				fbWriteEventData_Day(
					bExecute				:= bWriteData,
					sNetId					:= stFileSetupDayFile.sNetId,
					sPathName				:= stFileSetupDayFile.sTotalName,
					dwTransferBufferStartAdr:= dwTransferBufferStartAdr,
					iNewValues				:= (iIdx-1),
					udNumberofValues		:= udNumberofValues,
					udArrDataSize			:= udArrDataSize,
					udNumberOfEventDatas	:= udNumberOfEventDatas,
					sHeaderOfEventData		:= sHeaderOfEventData,
					eDataType				:= eDataType,
					bBusy					=> ,
					bDone					=> ,
					bError					=> bError,
					nErrId					=> nErrId );
				bWriteDayFileCopy		:= TRUE;
			ELSE
				bWriteDayFileCopy		:= FALSE;
			END_IF

			bWriteData := FALSE;
			state := 1;
		END_IF

		1:
		(* wait for the entries to be written *)
		fbWriteEventData( nNextPointerLoc:= nNextPointerLoc,);
		IF bWriteDayFileCopy THEN
			fbWriteEventData_Day( );
		END_IF
		IF NOT fbWriteEventData.bBusy
	           AND ( (bWriteDayFileCopy AND NOT fbWriteEventData_Day.bBusy) OR NOT bWriteDayFileCopy)
		    THEN
			fbWriteEventData( bExecute:= FALSE,nNextPointerLoc	:= nNextPointerLoc,);
			fbWriteEventData_Day(bExecute := FALSE);

			(*==========================================================*)
			(*  Counter for diagnostic   *)
			(*==========================================================*)
			rTrigErrorWriteData1(CLK:=fbWriteEventData.bError);
			IF rTrigErrorWriteData1.Q THEN
				iErrCounterEventData := iErrCounterEventData + 1;
			END_IF
			rTrigErrorWriteData2(CLK:=fbWriteEventData_Day.bError);
			IF rTrigErrorWriteData2.Q THEN
				iErrCounterEventData_Day := iErrCounterEventData_Day + 1;
			END_IF


			IF NOT fbWriteEventData.bBusy
			    AND ( (bWriteDayFileCopy AND NOT fbWriteEventData_Day.bError) OR NOT bWriteDayFileCopy)
	                  THEN
				(* discard the values already written in file from transfer buffer;
				    move the next values up to the first memory place [first place in the second memory part],make space for later entries *)
				udValuesNotWritten := iIdx-1-fbWriteEventData.udValuesWritten;
				MEMMOVE(
					dwTransferBufferStartAdr,
					dwTransferBufferStartAdr+(fbWriteEventData.udValuesWritten * iOneEntrySize) ,
					udValuesNotWritten * iOneEntrySize);
				(* clear the later space after the values are not written *)

				MEMSET(
					dwTransferBufferStartAdr+(udValuesNotWritten * iOneEntrySize),
					00,
					(udNumberofValues - 1 - udValuesNotWritten) * iOneEntrySize);

	iIdx := iIdx - UDINT_TO_INT(fbWriteEventData.udValuesWritten);
				state := 0;
			END_IF

			IF  NOT fbWriteEventData.bBusy AND NOT  fbWriteEventData.bBusy AND
		 	     NOT	fbWriteEventData.bError AND NOT fbWriteEventData_Day.bError THEN
				state := 0;
			ELSIF (fbWriteEventData.bError OR fbWriteEventData_Day.bError) THEN
				bError:=TRUE;
				state := 0;
			END_IF
		END_IF

	END_CASE


	(*==========================================================*)
	(*  Write to Novram  *)
	(*==========================================================*)
(*	IF NOT bInitNovRAM  AND gbEmbeddedHardwareDetected THEN											(*NEEDED?*)
	
		strucToNOVRAM.iRingBuffer_NextPointerLocation:= nNextPointerLoc;

	END_IF
*)
(*=========== END OF FUNCTION_BLOCK / PROGRAMM =============*)

ACTION M_AddEvent:
IF bInit THEN
	M1_Init( );
END_IF

(* Perform various checks *)
M2_Check( );

(* if no error and trigger event then add the entries *)
IF NOT bInitError AND bTrigEvent
THEN
	iNewValues := iNewValues + 1;		(* count the number of new entries added *)
	IF udCurrentAddIndex = 0 THEN
		udCurrentAddIndex := 1;			(* current index; where the newest entry is located *)
	ELSE
		udCurrentAddIndex := udCurrentAddIndex + 1;
		IF udCurrentAddIndex > udNumberofValues THEN (* current index; wrap around if max reached *)
			udCurrentAddIndex := 1;
		END_IF
	END_IF
	IF udCounter < udNumberOfValues THEN
		udUsedVal := udUsedVal + 1;			(* used index; the number of used entries; once udNumberOfValues reached remains constant to udNumberOfValues *)
	ELSE
		udUsedVal := udNumberofValues;
	END_IF

	IF udUsedVal < udNumberofValues THEN
		udOldestAddIndex := 1;				(* oldest index; wrap around if max reached *)
	ELSIF udUsedVal = udNumberofValues THEN
		udOldestAddIndex := udCurrentAddIndex + 1;
		IF udOldestAddIndex > udNumberofValues THEN		(* oldest index; where the oldest entry is located *)
			udOldestAddIndex := udOldestAddIndex - udNumberofValues;
		END_IF
	END_IF

(*========================================================================*)
(*		 limit description to    STRING[guiKeyAndTextLen];						   *)
(*		 max using length is [uiKeyAndTextLen - sKeySize]                                                     *)
(*=========================================================================*)
	sKeyAndText 			:= CONCAT(sTrigEventKey,'   ');  (* 3 spaces *)
	uiLENsTrigEventText 	:= LEN(sTrigEventText);
	uiLENsMaxText 		:= SIZEOF(sTrigEventText) - LEN(sKeyAndText);
	IF (uiLENsTrigEventText>uiLENsMaxText) THEN
		sTrigEventText := MID(sTrigEventText,0,uiLENsMaxText);
	END_IF
	sKeyAndText := CONCAT(sKeyAndText,sTrigEventText);

	iAddOffset := UDINT_TO_INT(udCurrentAddIndex-1) * iOneEntrySize; (* calculate the offset to be added according to the current index number *)

(*========================================================================*)
(*     fuse the key and text for trigger event together into one string, copy other values        *)
(*========================================================================*)
	(* Add the entry into the buffer *)
	(* Timestamp ------------------------------------- *)

	MEMCPY(dwBufferStartAdr + iAddOffset,ADR(sTimeStamp),SIZEOF(sTimeStamp));
	iSizeOf 			:= SIZEOF(sTimeStamp);
	iAddOffset 		:= iAddOffset + iSizeOf;
	uiCheckEntryLength:= iSizeOf; 					(* check entry length *)

	(* Key and the description -------------------- *)
	MEMCPY(dwBufferStartAdr + iAddOffset,ADR(sKeyAndText),SIZEOF(sKeyAndText));
	iSizeOf 			:= SIZEOF(sKeyAndText);
	iAddOffset 		:= iAddOffset + iSizeOf;
	uiCheckEntryLength:= uiCheckEntryLength + iSizeOf; 	(* check entry length *)

	(* User name --------------------------------------- *)
	MEMCPY(dwBufferStartAdr + iAddOffset,ADR(sUserName),SIZEOF(sUserName));
	iSizeOf 			:= SIZEOF(sUserName);
	iAddOffset 		:= iAddOffset + iSizeOf;
	uiCheckEntryLength:= uiCheckEntryLength + iSizeOf; 	(* check entry length *)

	(* Brake program --------------------------------------- *)
	MEMCPY(dwBufferStartAdr + iAddOffset,ADR(sBrakeProgram),SIZEOF(sBrakeProgram));
	iSizeOf 			:= SIZEOF(sBrakeProgram);
	iAddOffset 		:= iAddOffset + iSizeOf;
	uiCheckEntryLength:= uiCheckEntryLength + iSizeOf; 	(* check entry length *)



(*========================================================================*)
(*				 process value for logging only for real-type                                                  *)
(*=========================================================================*)
	(* copy the event datas into memory *)
	FOR i := 1 TO iNumberOfEventDatas DO

		CASE eDataType[i] OF
			(* Delete other type of data*)


			eReal :

				MEMCPY(dwBufferStartAdr + iAddOffset, dwArrDataAdr[i], udArrDataSize[i]);
				ar_iAddOffset[i] := iAddOffset;
				iAddOffset := iAddOffset + UDINT_TO_INT(udArrDataSize[i]);

		END_CASE


		iSizeOf 		:= UDINT_TO_INT(udArrDataSize[i]);
		uiCheckEntryLength:= uiCheckEntryLength + iSizeOf; 	(* check entry length *)

	END_FOR

(*========================================================================*)
(*				 Check length of data and the buffer entry size in the array		              *)
(*=========================================================================*)
	IF (uiCheckEntryLength>iOneEntrySize ) THEN
		uiCheckLenghtError := uiCheckLenghtError + 1;
		strLastKeyError := sKeyAndText;
	END_IF

	bCheck := TRUE;
END_IF
END_ACTION

ACTION M_CheckEvent:
(* At the end of the PLC cycle Check the data and order in ascending sequence *)
IF bCheck THEN (* bcheck is set to true by M_AddEvent; which means when no events or M_AddEvent not called, no data exists and hence no check performed *)

	iNumberOfValues := UDINT_TO_INT(udNumberofValues);		(* copy udint into int form *)

	(* if fill the buffer from beginning then reset the whole buffer *)
	IF iIdx = 1 THEN
		MEMSET(dwTransferBufferStartAdr,00,udSizeOfeachBlock);		(* reset the buffer *)
	END_IF

	(* see if all the new values fit into transfer buffer, else reassign New values to fitting number of values *)
	IF (iIdx + iNewValues) > (iNumberOfValues - 1) THEN
		iNewValues := (iNumberOfValues - 1) - iIdx;
	END_IF

	(* Copy the entries into transfer buffer *)
	IF udCurrentAddIndex >= iNewValues THEN 				(* If current index went once round the ring and is less then the new events added, which means some new events at the end of Ring Buffer and some in the beginning *)
		(* if New values are less than the current index that means all the values are in the beginning *)
		MEMCPY(
			dwTransferBufferStartAdr+((iIdx-1)*iOneEntrySize),
			dwBufferStartAdr+((udCurrentAddIndex - iNewValues)*iOneEntrySize),
			iNewValues*iOneEntrySize);


	ELSE
		(* if new values is greater than the current index that means some are at the end and rest in the beginning of the bufffer *)
		udOldValuesToBeCopied := iNewValues - udCurrentAddIndex;

		MEMCPY(
			dwTransferBufferStartAdr+((iIdx-1)*iOneEntrySize),
			dwBufferStartAdr+((udNumberofValues - udOldValuesToBeCopied)*iOneEntrySize),
			udOldValuesToBeCopied*iOneEntrySize);

		MEMCPY(
			dwTransferBufferStartAdr+((iIdx-1+udOldValuesToBeCopied)*iOneEntrySize),
			dwBufferStartAdr,
			udCurrentAddIndex*iOneEntrySize);
	END_IF

(*========================================================================*)
(*                                                      to sort out key number                                                                      *)
(*========================================================================*)
(*																									(*WIESO ausgeklammert?*)
	jIdx := iIdx;
	FOR i := iIdx TO (iIdx - 1 + iNewValues) DO		(* for loop from new index value to the number of new values *)

		MEMCPY(
			ADR(sKeyAndText_1),
			dwTransferBufferStartAdr+((i-1)*iOneEntrySize)+ SIZEOF(sTimeStamp),
			SIZEOF(sTrigEvent));

		sKeyAndText_1 := LEFT (sKeyAndText_1,(FIND(sKeyAndText_1,'   '))-1); (*01_05_001*)
		sKeyAndText_1 := DELETE (sKeyAndText_1,1,3);(*0105_001*)
		sKeyAndText_1 := DELETE (sKeyAndText_1,1,5); (*0105001*)
		udKeyAndText_1 := STRING_TO_UDINT(sKeyAndText_1);
		(* Arrange the key in an ascending order *)
		FOR j := jIdx TO (jIdx -1 + iNewValues) DO
			MEMCPY(
				ADR(sKeyAndText_2),
				dwTransferBufferStartAdr+((j-1)*iOneEntrySize)+SIZEOF(sTimeStamp),
				SIZEOF(sTrigEvent));

			sKeyAndText_2 := LEFT (sKeyAndText_2,(FIND(sKeyAndText_2,'   '))-1); (*01_05_001*)
			sKeyAndText_2 := DELETE (sKeyAndText_2,1,3);(*0105_001*) (* delete underscore *)
			sKeyAndText_2 := DELETE (sKeyAndText_2,1,5); (*0105001*) (* delete underscore *)
			udKeyAndText_2 := STRING_TO_INT(sKeyAndText_2);	(* convert string to a number for the necessary checks to sort *)
			IF udKeyAndText_1 < udKeyAndText_2 THEN
				(* use last memory address as temp memory space for comparison *)
				MEMCPY(
					dwTransferBufferStartAdr+((iNumberOfValues-1)*iOneEntrySize),
					dwTransferBufferStartAdr+((j-1)*iOneEntrySize),
					iOneEntrySize);
				MEMCPY(
					dwTransferBufferStartAdr+((j-1)*iOneEntrySize),
					dwTransferBufferStartAdr+((i-1)*iOneEntrySize),
					iOneEntrySize);
				MEMCPY(
					dwTransferBufferStartAdr+((i-1)*iOneEntrySize),
					dwTransferBufferStartAdr +((iNumberOfValues-1)*iOneEntrySize),
					iOneEntrySize);

				udKeyAndText_1 := udKeyAndText_2;			(*exchange the strings *)
			END_IF
		END_FOR
	END_FOR
	(*========================================================================*)
	(*                                                 end  to sort out key number                                                                  *)
	(*========================================================================*)
*)
	bCheck := FALSE;			(* Checking done *)
	iIdx := iIdx + iNewValues;	(* calculate where the index stands; increment the value of index by number of new values *)

	iEntriesWritten := iEntriesWritten + iNewValues;		(* Count the number of entries written *)
	IF iEntriesWritten > udNumberofValues THEN				(* If overflow then calculate relative count *)
		iEntriesWritten := UDINT_TO_INT(udNumberofValues - INT_TO_UDINT(iEntriesWritten));
	END_IF

	IF (iIdx-1) > 0 AND state = 0 THEN
		bWriteData := TRUE;
	END_IF
	iNewValues := 0;				(* reset the new values counter to zero *)

END_IF
END_ACTION

ACTION M1_Init:
bInit := FALSE;

iOneEntrySize := 0;				(* size of event in memory *)
iOneEntrySize := 	SIZEOF(sTimeStamp)+
				SIZEOF(sTrigEventText)+  (*before sTrigEvent*)
					SIZEOF(sUserName) +
					SIZEOF(sBrakeProgram);

iOneEntryLength := 0;			(* length of the event when written in file *)
iOneEntryLength :=	SIZEOF(sTimeStamp) +
					LEN(sTab) +
				SIZEOF(sTrigEventText)+  (*before SIZEOF(sTrigEventKey) + SIZEOF(sTrigEventText)+*)
					LEN(sTab) +
					SIZEOF(sUserName) +
					LEN(sTab) +
					SIZEOF(sBrakeProgram) +
					LEN(sTab);

iNumberOfEventDatas := UDINT_TO_INT(udNumberOfEventDatas);

(* Check the data type of all the required event datas; calculate entry length and size accordingly *)
FOR i := 1 TO iNumberOfEventDatas DO
	CASE eDataType[i] OF
		eBool :
			iOneEntryLength := iOneEntryLength + 5;			(* when converted into string *)
			iOneEntrySize := iOneEntrySize +  UDINT_TO_INT(udArrDataSize[i]);

		eReal :
			iOneEntryLength := iOneEntryLength + 17;		(* when converted into string *)
			iOneEntrySize := iOneEntrySize +  UDINT_TO_INT(udArrDataSize[i]);

	END_CASE
	IF i < udNumberOfEventDatas THEN
		iOneEntryLength := iOneEntryLength + LEN(sTab);	(* calculate the tabs too into the length of string *)
	ELSE
		iOneEntryLength := iOneEntryLength + LEN(sLineFeed);	(* calculate the linefeed too into the length of string *)
	END_IF

END_FOR

IF ((udLoggedEventSize/2) MOD iOneEntrySize) = 0 THEN		(* Check if all the data fits into the given memory block *)
	udSizeOfeachBlock := udLoggedEventSize/2;
	udNumberofValues := udLoggedEventSize/ (iOneEntrySize *2);	(* calculate the number of events that can be logged *)
	(* calulate the start and end addresses of the buffer *)
	dwBufferStartAdr := dwLoggedEventAdr;
	dwBufferEndAdr	:= dwLoggedEventAdr + udLoggedEventSize/2;
	dwTransferBufferStartAdr := dwBufferEndAdr;
	dwTransferBufferEndAdr := dwLoggedEventAdr + udLoggedEventSize;
ELSE
	bInitError := TRUE;	(* size not appropriate *)
	nErrId := 1;
END_IF
END_ACTION

ACTION M2_Check:
(* check if the file path is given *)
IF LEN(stFileSetup.sPathName)= 0
THEN
	ADSLOGSTR( 	msgCtrlMask := ADSLOG_MSGTYPE_WARN,
				msgFmtStr := 'PLC Msg: FilePath is empty; %s',
				strArg := stFileSetup.sPathName);
	RETURN;
END_IF
(* check if the file path is given for Day file *)
IF bWriteDayFile AND LEN(stFileSetupDayFile.sPathName)= 0
THEN
	ADSLOGSTR( 	msgCtrlMask := ADSLOG_MSGTYPE_WARN,
				msgFmtStr := 'PLC Msg: FilePath_DayFile is empty; %s',
				strArg := stFileSetupDayFile.sPathName);
	RETURN;
END_IF
(* If same file name for RingBufferFile and for EventDayFile *)
IF bWriteDayFile AND (stFileSetup.sPathName = stFileSetupDayFile.sPathName)
THEN
	ADSLOGSTR( 	msgCtrlMask := ADSLOG_MSGTYPE_WARN,
				msgFmtStr := 'PLC Msg: Same file path given; %s',
				strArg := stFileSetupDayFile.sPathName);
	RETURN;
END_IF

(* Check the start, end addresses of buffers *)
IF dwBufferStartAdr = 0 OR dwBufferEndAdr = 0 OR
   dwTransferBufferStartAdr = 0 OR dwTransferBufferEndAdr = 0
THEN
	ADSLOGDINT( msgCtrlMask := ADSLOG_MSGTYPE_WARN,
				msgFmtStr := 'PLC Msg: Buffer Size does not match; Buffer Addresses zero; %s',
				dintArg := MIN(dwBufferStartAdr,MIN(dwBufferEndAdr,MIN(dwTransferBufferStartAdr,dwTransferBufferEndAdr))));
	RETURN;
END_IF

(* If entry length in file larger than 255, string operations like CONCAT, LEN do not work *)
IF iOneEntryLength > 255
THEN
	ADSLOGDINT( msgCtrlMask := ADSLOG_MSGTYPE_WARN,
				msgFmtStr := 'PLC Msg: Entry of one event is greater 255; %s',
				dintArg := iOneEntryLength);
	RETURN;
END_IF

(* Check the entry size in memory *)
IF iOneEntrySize = 0
THEN
	ADSLOGDINT( msgCtrlMask := ADSLOG_MSGTYPE_WARN,
				msgFmtStr := 'PLC Msg: Buffer size is Zero; %d',
				dintArg := iOneEntrySize);
	RETURN;
END_IF

(* Check if the trigger event key is not empty *)
IF sTrigEventKey = ''
THEN
	ADSLOGSTR( 	msgCtrlMask := ADSLOG_MSGTYPE_WARN,
				msgFmtStr := 'PLC Msg: TrigEventKey is empty; %s',
				strArg := sTrigEventKey);
	RETURN;
END_IF

(* Check if the trigger event key is according to the format*)
IF LEN(sTrigEventKey) < SIZEOF(sTrigEventKey)-1
THEN
	ADSLOGSTR( 	msgCtrlMask := ADSLOG_MSGTYPE_WARN,
				msgFmtStr := 'PLC Msg: TrigEventKey length not as per defined; %s',
				strArg := sTrigEventKey);
	RETURN;
END_IF

(* Check if the Buffer start address is not zero; nonassigned *)
IF dwBufferStartAdr = 0
THEN
	ADSLOGSTR( 	msgCtrlMask := ADSLOG_MSGTYPE_WARN,
				msgFmtStr := 'PLC Msg: Buffer start address is 0; %s',
				strArg := sTrigEventKey);
	RETURN;
END_IF

(* Check if the Buffer end address is not zero; nonassigned *)
IF dwBufferEndAdr = 0
THEN
	ADSLOGSTR( 	msgCtrlMask := ADSLOG_MSGTYPE_WARN,
				msgFmtStr := 'PLC Msg: Buffer end address is 0; %s',
				strArg := sTrigEventKey);
	RETURN;
END_IF

(* Check if the transfer Buffer start address is not zero; nonassigned *)
IF dwTransferBufferStartAdr = 0
THEN
	ADSLOGSTR( 	msgCtrlMask := ADSLOG_MSGTYPE_WARN,
				msgFmtStr := 'PLC Msg: Buffer start address is 0; %s',
				strArg := sTrigEventKey);
	RETURN;
END_IF

(* Check if the transfer Buffer end address is not zero; nonassigned *)
IF dwTransferBufferEndAdr = 0
THEN
	ADSLOGSTR( 	msgCtrlMask := ADSLOG_MSGTYPE_WARN,
				msgFmtStr := 'PLC Msg: Buffer end address is 0; %s',
				strArg := sTrigEventKey);
	RETURN;
END_IF

(* Check if the size of block is nonzero; nonassigned *)
IF udSizeOfeachBlock = 0
THEN
	ADSLOGSTR( 	msgCtrlMask := ADSLOG_MSGTYPE_WARN,
				msgFmtStr := 'PLC Msg: Buffer size is 0; %s',
				strArg := sTrigEventKey);
	RETURN;
END_IF
END_ACTION

END_FUNCTION_BLOCK

// ---- Alarm System/POUs/02_Alarm_Handling/FB_WriteEventData.TcPOU
FUNCTION_BLOCK FB_WriteEventData
(**********************************************************************************)
(**********************************************************************************)
(*  	VERSION:			002.012
							                									
	PROGRAMMED BY:	Puja					  					
  	Changed by:			Hardy Patommel							
*)  																		
(*-----------------------------------------------------------------------------------------------------------------------------------*)
(*  REVISIONS:						                							 
   	Date		|	Version/Author 	|	Remark
	----------------------------------------------------------------------------------------------------
	2007-10-08	|	001.001     HP		|   	formatting the REAL value FOR the file output
	2008-03-04	|	002.000     HP		|   	add header function block
	2008-03-27	|	002.001     HP		|   	add header length with initialization value
	2009-03-26	|	002.010     HP		|   	get header length as parameter
	2009-03-27	|	002.011     HP		|   	change strBuffer size with a constant variable
	2009-08-09	|	002.012     HP		|   	change sTimestamp[24]
*)
(*-----------------------------------------------------------------------------------------------------------------------------------*)
(*  	DESCRIPTION:
	Constant value for the file layout >>	
		nNextPointerLoc			: DINT;		>>> actual position for the next entry [NOVRAM]
		iFirstHeaderLEN1			: INT:=1000;	>>> header size without column-description

	Note:
		 iFirstHeaderLEN and iColumnLineLEN are only necessary when the data file will be create
*)
(**********************************************************************************)
(**********************************************************************************)
VAR_INPUT
	bExecute 				: BOOL;
	sNetId					: T_AmsNetId;
	sPathName				: T_MaxString;
	dwTransferBufferStartAdr	: DWORD;
	iNewValues				: INT;
	udNumberofValues 		: UDINT;
	udNumberOfEventDatas	: UDINT;
	udArrDataSize			: ARRAY [1..NUMBER_OF_EVENT_DATAS] OF UDINT;
	eDataType				: ARRAY [1..NUMBER_OF_EVENT_DATAS] OF E_DataType;
	sHeaderOfEventData	: ARRAY [1..giGeneralLoggerChannelInUsed] OF STRING(giGeneralLenghtOfName);
	iHeaderLEN				: INT;  (*length of whole header; first header + column*)
END_VAR
VAR_IN_OUT
	nNextPointerLoc			: DINT;
END_VAR
VAR_OUTPUT
	udValuesWritten			: UDINT;
	bBusy					: BOOL;
	bDone					: BOOL;
	bError					: BOOL;
	nErrId					: UDINT;
END_VAR
VAR
	RExec_Trig				: R_TRIG;
	hFile					: UINT;
	fbFileOpen				: FB_FileOpen;
	fbFileSeek				: FB_FileSeek;
	fbFileWrite				: FB_FileWrite;
	fbFileClose				: FB_FileClose;
	tAdsTimeOut			: TIME:= T#10s;
	eFileState				: E_FileState_SC;
	nMode					: DWORD;
	sStrBuffer				: STRING(guiStrBufferSize);	(* header 1100 + row 200 * 218 sign = 44700*)
	sStrHeader				: STRING(2170);	 	(*10 row with 217 sign*)
	sVar					: STRING(255);
	sHeader					: STRING(giHeaderColumnLineLEN); (*:='TimeStampUTC$TTrigKey$TUserName$TBrakeProgram$T'; (*!!HP*)		DISABLED BY NIHAL MALIK *)
	sTab					: STRING[2] := '$T';
	sLineFeed				: STRING[4] := '$R$N';

	i						: INT;


	dwCaptureTransferBufferStartAdr : DWORD;
	sTimeStamp			: STRING[24];	(* Time the Statuscode becomes true *)
	sTrigEvent				: STRING[guiKeyAndTextLen];	(* key and Text of Statuscode, like sKeyAndText[80] in M_AddEvent*)
	sUserName				: STRING[24];	(* name of the user who had the Active Status to do the operation *)
	sBrakeProgram			: STRING[4]; 	(* Activated brake program *)
	rVar						: REAL;
(*	eTime					:= 12,
	eDate					:= 13,
	eTime_OF_Day			:= 14,
	eDateAndTime			:= 15,
	eString					:= 16,	*)
	iCopyOffset				: INT;

	iPrepIndex				: INT;
	iStrBufferIdx				: UINT; (*Index buffer*)

	iStrLineIdx				: INT; (*Index line*)
	iStuff					: INT;
	iStartStuffIndex			: INT;
	iEndStuffIndex			: INT;
	iStartIndex				: INT;
	iEndIndex				: INT;

	iBatchValue				: INT := 20;(* in batch of how many entries is the data to be written *)
	iEventsWrittenCurrent		: INT;		(* Event written in current cycle *)
	iCaptureNewValues		: INT;		(* captures new values *)
	iEntriesWritten			: INT;		(* Entries Written; so as to calculate the next pointer location*)
	iFittingEntries				: INT;		(* number of entries fitting *)
	iEventsInCycle			: INT;		(* In how many batches is data written *)
	bHeader					: BOOL;		(* If a new file write then to write the header *)
	iCounter					: INT;		(* Total number of entries written till now, so as to tally *)
	iNumberOfEventDatas		: INT;
	sTimestampShort			: STRING[12];
	sRealDataReduce		: STRING[10];
	iLength					: INT;
	iDiffenzLength				: INT;
	iForIndex					: UINT;

	fbHeaderForLogging		: FB_HeaderForLogging;
	iFirstHeaderLEN			: INT;
	iColumnLineLEN		: INT;
	uiCountsOfLine			: UINT;
	udiCheckHeaderLength	: UDINT;

END_VAR

(*========== START OF FUNCTION_BLOCK / PROGRAMM ============*)


(*=====================================================================*)
(*					write event data to file        							     *)
(*=====================================================================*)
RExec_Trig( CLK := bExecute );

CASE eFileState OF
   eInit_SC:
		IF RExec_Trig.Q THEN	(* Rising edge triggered *)
			bBusy 	:= TRUE;
			bError	:= FALSE;
			bDone 	:= FALSE;
			nErrId	:= 0;
			hFile	:= 0;

			dwCaptureTransferBufferStartAdr := dwTransferBufferStartAdr;(* capture the transfer buffer address *)
			iCaptureNewValues	:= iNewValues;					(* make a copy of the input newvalues *)
			iNumberOfEventDatas := UDINT_TO_INT(udNumberOfEventDatas);
			nMode := FOPEN_MODEREAD OR FOPEN_MODEPLUS OR FOPEN_MODEBINARY;
			(*nMode := FOPEN_MODEAPPEND OR FOPEN_MODEPLUS OR FOPEN_MODEBINARY;*)
			iBatchValue := (guiStrBufferSize/iOneEntryLength) - 1;		(* calculate the batch size in which data is to be written *)
			IF iCaptureNewValues > 0 THEN
				sTimestampShort :='4';(* FUN_TimeToString(Lib_strucSystemTime); (*access time *)TO ACTION*)
				(* Open a file *)
				fbFileOpen( bExecute	:= FALSE	);
				fbFileOpen(	bExecute	:= TRUE,
							sNetId		:= sNetID,
							sPathName	:=sPathName,
							nMode		:= nMode,
							ePath		:= Path_Generic,
							tTimeout	:= tAdsTimeOut );

				eFileState := eFileOpen_SC;
				(* reset the variables *)
				iStartIndex := 1;
				iStrBufferIdx := 0;
				sStrBuffer := '';
				sVar := '';
				udValuesWritten := 0;
			END_IF
		END_IF

		g_TriggSendExeAlarmList := FALSE;

	eFileOpen_SC:	(* Wait for the file to be opened *)
		fbFileOpen( );
		IF NOT fbFileOpen.bBusy THEN
			fbFileOpen(	bExecute := FALSE);

			IF NOT fbFileOpen.bError THEN		(* if no error; File already exists *)

				IF NOT bHeader AND nNextPointerLoc > 0 THEN		(*Check the next pointer persistent value*)
					nNextPointerLoc := nNextPointerLoc -  iHeaderLEN;
					IF  iOneEntryLength <> 0 THEN
						iEntriesWritten := DINT_TO_INT(nNextPointerLoc/iOneEntryLength);
						iCounter := DINT_TO_INT(nNextPointerLoc/iOneEntryLength);
					END_IF

					nNextPointerLoc := nNextPointerLoc + iHeaderLEN;

				ELSIF bHeader THEN		(* if file did not exist then iEntriesWritten to beginning *)
					iEntriesWritten := 0;
					iCounter := 0;
				ELSIF NOT bHeader AND (nNextPointerLoc = 0) THEN	(* reset all and file exist *)
					nNextPointerLoc := nNextPointerLoc + iHeaderLEN;
				END_IF
				iFittingEntries := UDINT_TO_INT(udNumberofValues)  - iEntriesWritten ;
				(* calculate the minimum of Captured values, Batch value and how many can fit *)
				iEndIndex := MIN(iCaptureNewValues,iBatchValue);
				iEventsWrittenCurrent := iEndIndex := MIN(iEndIndex, iFittingEntries);

				hFile  := fbFileOpen.hFile;
				fbFileSeek( bExecute := FALSE);			(* File Seek *)
				fbFileSeek(	sNetId 		:= sNetId,
							hFile		:= hFile,
							nSeekPos	:= nNextPointerLoc,			(* File pointer to zero *)
							eOrigin		:= SEEK_SET,
							bExecute	:= TRUE,
							tTimeout	:= tAdsTimeOut,
							);
				eFileState := eFileSeek_SC;

			ELSE	(*if error, File does not exist; a new file is to be written *)

				(*create new file with header*)
				nMode := FOPEN_MODEWRITE  OR FOPEN_MODEPLUS OR FOPEN_MODEBINARY;
				(*nMode := FOPEN_MODEAPPEND  OR FOPEN_MODEPLUS OR FOPEN_MODEBINARY;*)
				fbFileOpen( bExecute	:= FALSE	);
				fbFileOpen(	bExecute	:= TRUE,
				 			sNetId		:= sNetID,
							sPathName	:= sPathName,
							nMode		:= nMode,
							ePath		:= Path_Generic,
							tTimeout	:= tAdsTimeOut );
				eFileState := eFileOpen_SC;
				nNextPointerLoc := 0;
				iCounter := 0;
				(* if new file is being written then write down the header *)
				bHeader := TRUE;

				fbHeaderForLogging(
						st_TurbineIdent		:= st_xTurbineIdent ,			(*general machine info*)
						s_FileDescription	:= fbSCLogger.stFileSetup.sFileDescription,
						s_ColumnText 		:= gstrRingBufferFileColumnText,
						ar_ColumnText		:= sHeaderOfEventData,		(*array of column description*)
						iCountsOfColumns	:= iNumberOfEventDatas,	(*counts of columns*)
						iOneEntryLength	:= giRingBufferFileOneEntryLength,(*length of every entry, all lines with the same length, see init-logger*)
				//ACTION		adr_sHeader1		:= ADR(sStrHeader) ,		(*part one of the header*)
				//ACTION		adr_sColumnLine	:= ADR(sHeader),			(*part two of the header*)
						iCountsOfLine		=> uiCountsOfLine,			(*lines of the part one header*)
						iHeaderLEN			=> iFirstHeaderLEN,			(*length of the part one header*)
						iColumnLineLEN	=> iColumnLineLEN);		(*length of the part two header*)


				(*Check the header length: header and column-description*)
				udiCheckHeaderLength := LEN(sStrHeader) + LEN(sHeader);
			END_IF
		END_IF


	eFileSeek_SC:
		fbFileSeek( );
		IF NOT fbFileSeek.bBusy THEN
			fbFileSeek(bExecute := FALSE );
			IF NOT fbFileSeek.bError THEN

				(* Prepare the data to be written *)
				M_PrepareWriteData( );

				(* Write into File *)
				fbFileWrite( 	bExecute	:= FALSE	);
				fbFileWrite(  	bExecute	:= TRUE,
								sNetId		:= sNetID,
								hFile		:= hFile,
								pWriteBuff	:= ADR(sStrBuffer),
								cbWriteLen	:= iStrBufferIdx,         (*Write not the whole Buffer, only new entries*)
								tTimeout	:= tAdsTimeOut	);

				iStrBufferIdx := iStrBufferIdx;

				eFileState := eFileWrite_SC;

			ELSE
				bBusy := FALSE;
				bError := TRUE;
				nErrId := fbFileSeek.nErrId;
				eFileState := eInit_SC;
			END_IF
		END_IF


	eFileWrite_SC:	(* Wait until  the file is written *)
		fbFileWrite();
		IF NOT fbFileWrite.bBusy THEN
			fbFileWrite(bExecute := FALSE);
			IF NOT fbFileWrite.bError THEN
				bHeader := FALSE;
				IF iCaptureNewValues > iEventsWrittenCurrent THEN		(* data is to be written into two or more parts *)
					IF iEventsWrittenCurrent = iBatchValue THEN
						(* sStrBuffer was insufficient to occupy all entries, Fitting entries were greater than that, continue writting at same file pointer *)
						iEntriesWritten := iEntriesWritten + iBatchValue;
						iFittingEntries := iFittingEntries - iEventsWrittenCurrent;
						iCaptureNewValues := iCaptureNewValues - iEventsWrittenCurrent;
						iEndIndex := MIN( iCaptureNewValues , iBatchValue);
						iEventsWrittenCurrent := iEndIndex := MIN( iEndIndex , iFittingEntries); (* Events to be written in current write cycle;*)
						iStrBufferIdx := 0;				(* reset while new batch write *)

						(* Prepare the next batch of data to be written *)
						M_PrepareWriteData( );

						(* Write into File *)
						fbFileWrite( 	bExecute	:= FALSE	);
						fbFileWrite(  	bExecute	:= TRUE,
								sNetId		:= sNetID,
								hFile		:= hFile,
								pWriteBuff	:= ADR(sStrBuffer),
								cbWriteLen	:= iStrBufferIdx,         (*Write not the whole Buffer, only new entries*)
								tTimeout	:= tAdsTimeOut	);

						iStrBufferIdx := iStrBufferIdx;
						eFileState := eFileWrite_SC;

					ELSIF iEventsWrittenCurrent = iFittingEntries THEN
						(* if the events written was just fit; pointer location to be set to beginning of file *)
						(* -------------------------------------------------------------------------------------------------------------*)
						iEntriesWritten := 0;
						iFittingEntries := UDINT_TO_INT(udNumberofValues);		(* go to beginning of file and initialise fitting entries to max *)
						iCaptureNewValues := iCaptureNewValues - iEventsWrittenCurrent;
						iEventsWrittenCurrent := iEndIndex := MIN( iCaptureNewValues , iBatchValue);
						iStrBufferIdx := 0;

						(* calculate the next pointer location *)
						nNextPointerLoc := iHeaderLEN + (iEntriesWritten * iOneEntryLength);
						fbFileSeek( bExecute := FALSE);			(* File Seek *)
						fbFileSeek(	sNetId 		:= sNetId,
									hFile		:= hFile,
									nSeekPos	:= nNextPointerLoc,	(* File pointer to next loc - first line in file*)
									eOrigin		:= SEEK_SET,
									bExecute	:= TRUE,
									tTimeout	:= tAdsTimeOut
									);
						eFileState := eFileSeek_SC;
					END_IF

				ELSE	(* if exact fit then reintialise pointer to start of file *)
						(* ------------------------------------------------------------------*)
					IF iFittingEntries = iCaptureNewValues THEN
						iEntriesWritten := 0; (* actually 200 but reset to 1 *)
					ELSE
						iEntriesWritten := iEntriesWritten + iCaptureNewValues;
					END_IF
					nNextPointerLoc :=iHeaderLEN + ( iEntriesWritten * iOneEntryLength);
					(* Close the File *)
					fbFileClose(	bExecute:= FALSE	);
					fbFileClose(	bExecute:= TRUE,
									sNetId	:= sNetID,
									hFile	:= hFile,
									tTimeout:= tAdsTimeOut	);
					eFileState := eFileClose_SC;
				END_IF
			ELSE
				bBusy := FALSE;
				bError := TRUE;
				nErrId := fbFileWrite.nErrId;
				eFileState := eInit_SC;
			END_IF
		END_IF



	eFileClose_SC:	(* Wait untill File is closed *)
		fbFileClose();
		IF NOT fbFileClose.bBusy THEN
			fbFileClose( bExecute:= FALSE );
			IF NOT fbFileClose.bError THEN
				IF iCounter >= UDINT_TO_INT(udNumberOfValues) THEN
					iCounter := iCounter;
				END_IF
				(*eFileState := eInit_SC;*)
				eFileState := eFileCopy_SC;
				bBusy  := FALSE;
				bDone  := TRUE;
				bHeader := FALSE;
				sStrBuffer := '';
				iCaptureNewValues := 0;
				iEventsInCycle := 0;
			ELSE
				bBusy := FALSE;
				bError := TRUE;
				nErrId := fbFileClose.nErrId;
				eFileState := eInit_SC;
			END_IF
		END_IF

		eFileCopy_SC:
			g_TriggSendExeAlarmList := TRUE;
			eFileState := eInit_SC;

END_CASE

(*=========== END OF FUNCTION_BLOCK / PROGRAMM =============*)

ACTION M_PrepareWriteData:
MEMSET(ADR(sStrBuffer) , 0, LEN(sStrBuffer));
IF bHeader  THEN
	(*Header part one*)
	MEMCPY(ADR(sStrBuffer) ,ADR(sStrHeader),iFirstHeaderLEN);
	(*Header part two, column description*)
	MEMCPY(ADR(sStrBuffer)+iFirstHeaderLEN ,ADR(sHeader),iColumnLineLEN);
	(*index for buffer entry after the header; iHeaderLEN := iFirstHeaderLEN + iColumnLineLEN;*)
	iStrBufferIdx := iHeaderLEN;
	(* Write into File *)
END_IF

(* Stuff the data to be written into a string buffer *)
FOR iPrepIndex := iStartIndex  TO iEndIndex DO	(* for loop from new index value to the number of new values *)
	iCopyOffset := (((iPrepIndex-1)+iEventsInCycle)*iOneEntrySize); (*iCopyOffset := Offset in array ringbuffer*)
	sVar := '';
	iStrLineIdx := 0; (*index for the line, function stuff line*)
	(*gets the new dataset ####################*)
	(*gets timestamp value ---------------*)
	MEMCPY(
		ADR(sTimeStamp),
		dwCaptureTransferBufferStartAdr+iCopyOffset,
		SIZEOF(sTimeStamp));
	sVar := CONCAT('',sTimeStamp);
	sVar := CONCAT(sVar,sTab);
	iCopyOffset := iCopyOffset + SIZEOF(sTimeStamp);

	(*gets trigger event string ---------------*)
	MEMCPY(
		ADR(sTrigEvent),
		dwCaptureTransferBufferStartAdr+iCopyOffset,
		SIZEOF(sTrigEvent));
	(*look and fill to 50 sign*)
	iLength := LEN(sTrigEvent);
	IF (iLength<giCountsOfKeyLetterForStatuscodeFile) THEN
		iDiffenzLength := giCountsOfKeyLetterForStatuscodeFile - iLength ;
		FOR iForIndex := 1 TO  iDiffenzLength DO
			sTrigEvent := CONCAT(sTrigEvent,' ');
		END_FOR
	END_IF
	sTrigEvent := sTrigEvent ;
	sVar := CONCAT(sVar,sTrigEvent);
	sVar := CONCAT(sVar,sTab);
	iCopyOffset := iCopyOffset + SIZEOF(sTrigEvent); (*read data out of log-array*)

	(*gets user name string ---------------*)
	MEMCPY(
		ADR(sUserName),
		dwCaptureTransferBufferStartAdr+iCopyOffset,
		SIZEOF(sUserName));
	sVar := CONCAT(sVar,sUserName);
	sVar := CONCAT(sVar,sTab);
	iCopyOffset := iCopyOffset + SIZEOF(sUserName);

	(*gets brake program string ---------------*)
	MEMCPY(
		ADR(sBrakeProgram),
		dwCaptureTransferBufferStartAdr+iCopyOffset,
		SIZEOF(sBrakeProgram));
	sVar := CONCAT(sVar,sBrakeProgram);
	sVar := CONCAT(sVar,sTab);
	iCopyOffset := iCopyOffset + SIZEOF(sBrakeProgram);

	(*gets configuration data  value ---------------*)
	(* convert appropriate event datas into string format and concat into one string buffer *)
	FOR i := 1 TO iNumberOfEventDatas DO
		CASE eDataType[i] OF

			eReal :
				(*formatting the real value*)
				MEMCPY(ADR(rVar),dwCaptureTransferBufferStartAdr+iCopyOffset,udArrDataSize[i]);
				sRealDataReduce := '8'(*FUN_Real_to_string(rVar,2)*);

				sVar := CONCAT(sVar,sRealDataReduce);
				sVar := CONCAT(sVar,sTab);	(* append tab *)
				iCopyOffset := iCopyOffset + UDINT_TO_INT(udArrDataSize[i]) ;

		END_CASE
	END_FOR


	iStrLineIdx := LEN(sVar);			(*length of string in one row, prepared for file logging*)
	iStartStuffIndex := iStrLineIdx + 1;		(*start address for stuff sign*)
	iEndStuffIndex := iOneEntryLength-2;

	(* append spaces to make every event of same length *)
	IF iStrLineIdx < iEndStuffIndex THEN
		FOR iStuff := iStartStuffIndex TO  iEndStuffIndex DO
			sVar := CONCAT(sVar,' ');
			iStrLineIdx := iStrLineIdx + 1;
		END_FOR
	END_IF
	sVar := CONCAT(sVar,sLineFeed);			(* append line feed *)
	iStrLineIdx := iStrLineIdx + LEN(sLineFeed);	(*length of string in one row*)

	(* copy the event into the string buffer *)
	IF bHeader THEN
		MEMCPY(
			ADR(sStrBuffer)+ iHeaderLEN + (iOneEntryLength * (iPrepIndex - 1)) ,
			ADR(sVar),
			iOneEntryLength);
	ELSE
		MEMCPY(
			ADR(sStrBuffer)+ (iOneEntryLength * (iPrepIndex - 1)) ,
			ADR(sVar),
			iOneEntryLength);
	END_IF

	iStrBufferIdx := iStrBufferIdx + iOneEntryLength;
	iStrLineIdx := 0;
	iCounter := iCounter + 1;


END_FOR

udValuesWritten := udValuesWritten + iEndIndex;	(* output how many values already written *)
iEventsInCycle := iEventsInCycle + iEndIndex;		(* Calculate the number of events written / in how many batches *)
END_ACTION

END_FUNCTION_BLOCK

// ---- Alarm System/POUs/02_Alarm_Handling/FB_HeaderForLogging.TcPOU
FUNCTION_BLOCK FB_HeaderForLogging
(**********************************************************************************)
(**********************************************************************************)
(*  	VERSION:			001.000
							                										
  	PROGRAMMED BY:	Hardy Patommel	  								
*)  																		
(*----------------------------------------------------------------------------------------------------------------------------*)
(*	Version history:														 *)
(*    	Date		|	Version/Author 	|	Remark
	----------------------------------------------------------------------------------------------------
	2008-03-03	|	001.000     HP		|	
	2008-03-07	|	001.001     HP		|	changed header building
	
						                								
*)
(*----------------------------------------------------------------------------------------------------------------------------*)
(*  	DESCRIPTION:
	combine the header for the log file e.g.

			1.	CompanyCode:	Name of comany
			2.	CountryCode:		xx
			3.	Flowfarm:		Flow energy park 24
			4.	TurbineNumber:	1
			5.	TurbineType:		123
			6.
			7.	Comment:	Statuscode ring buffer file
			8.
			9.
			10.	
			11.	TimeStampUTC				TrigKey	

*)
(**********************************************************************************)
(**********************************************************************************)
VAR_INPUT
	st_TurbineIdent			: ST_xTurbineIdent;	(*info structure*)
	s_FileDescription			: T_MaxString;
	s_ColumnText 			: T_MaxString;
(*	ar_ColumnText			: ARRAY [1..giNumberOf10minMeanChannels] OF STRING(giGeneralLenghtOfName);*)
	ar_ColumnText			: ARRAY [1..75] OF STRING(40);
	iCountsOfColumns 		: UINT;				(*counts of columns*)
	iOneEntryLength			: UINT; 				(*length of of entry*)
	adr_sHeader1			: DWORD; 			(*address of string: general description of machine, lenght = description + 6*255 *)
	adr_sColumnLine			: DWORD;	 		(*address of string: column description of table, lenght min.= 100*80 *)
END_VAR
VAR_OUTPUT
	iCountsOfLine				: UINT; 	(*counts of rows*)
	iHeaderLEN				: INT;	(*counts of byte*)
	iColumnLineLEN			: INT;	(*counts of byte*)
END_VAR
VAR
(*	sHeader					: STRING[giHeader1LEN]; 		*)		(*address of string: general description of machine, lenght = description + 6*255 *)
(*	sColumnLine				: STRING[giHeaderColumnLineLEN];	*)	(*address of string: column description of table, lenght min.= 100*80 *)

	sHeader					: STRING[1100]; 						(*address of string: general description of machine, lenght = description + 6*255 *)
	sColumnLine				: STRING[4096];						(*address of string: column description of table, lenght min.= 100*80 *)
	sTab					: STRING[2] := '$T';
	sLineFeed				: STRING[4] := '$R$N';
	sStrVar					: T_MaxString;
	sStrHeaderLine			: T_MaxString;
	udiStrWriteIndex			: UDINT;
	i: INT; (*for index*)

	iStrLEN: DINT;
	udiSize: UDINT;
END_VAR

(*=============== START OF FUNCTION_BLOCK / PROGRAMM ===============*)
	MEMSET(ADR(sHeader) , 0, LEN(sHeader));
	MEMSET(ADR(sColumnLine) , 0, LEN(sColumnLine));

(*=====================================================================*)
(*					HEADER PART 1 (general description)				     *)
(*=====================================================================*)
	iHeaderLEN 		:= 0;
	udiStrWriteIndex 	:= 0;
	(*Line: 1*)
	sStrHeaderLine 	:= '';
	sStrHeaderLine := CONCAT(sStrHeaderLine,'CompanyCode:');
	sStrHeaderLine := CONCAT(sStrHeaderLine,sTab);
	sStrHeaderLine := CONCAT(sStrHeaderLine, st_xTurbineIdent.sCompanyCode);

	iHeaderLEN := LEN(sStrHeaderLine);
	IF iHeaderLEN < giHeaderLineLenght THEN
		FOR i := iHeaderLEN+1 TO (giHeaderLineLenght-2) DO
			sStrHeaderLine := CONCAT(sStrHeaderLine,' ');		(* concat with stuff spaces *)
		END_FOR
	END_IF
	sStrHeaderLine := CONCAT(sStrHeaderLine,sLineFeed); (* concat Linefeed *)
	udiSize :=  LEN(sStrHeaderLine);
	MEMCPY( ADR(sHeader)+udiStrWriteIndex, ADR(sStrHeaderLine),udiSize);
	udiStrWriteIndex := udiStrWriteIndex + udiSize;

	(*Line: 2*)
	sStrHeaderLine 	:= '';
	sStrHeaderLine := CONCAT(sStrHeaderLine,'CountryCode:');
	sStrHeaderLine := CONCAT(sStrHeaderLine,sTab);
	sStrHeaderLine := CONCAT(sStrHeaderLine, UINT_TO_STRING(st_xTurbineIdent.byCountryCode));

	iHeaderLEN := LEN(sStrHeaderLine);
	IF iHeaderLEN < giHeaderLineLenght THEN
		FOR i := iHeaderLEN+1 TO (giHeaderLineLenght-2) DO
			sStrHeaderLine := CONCAT(sStrHeaderLine,' ');		(* concat with stuff spaces *)
		END_FOR
	END_IF
	sStrHeaderLine := CONCAT(sStrHeaderLine,sLineFeed); (* concat Linefeed *)
	udiSize :=  LEN(sStrHeaderLine);
	MEMCPY( ADR(sHeader)+udiStrWriteIndex, ADR(sStrHeaderLine),udiSize);
	udiStrWriteIndex := udiStrWriteIndex + udiSize;

	(*Line: 3*)
	sStrHeaderLine 	:= '';
	sStrHeaderLine := CONCAT(sStrHeaderLine,'Flowfarm:');
	sStrHeaderLine := CONCAT(sStrHeaderLine,sTab);
	sStrHeaderLine := CONCAT(sStrHeaderLine,st_xTurbineIdent.sFlowfarm);

	iHeaderLEN := LEN(sStrHeaderLine);
	IF iHeaderLEN < giHeaderLineLenght THEN
		FOR i := iHeaderLEN+1 TO (giHeaderLineLenght-2) DO
			sStrHeaderLine := CONCAT(sStrHeaderLine,' ');		(* concat with stuff spaces *)
		END_FOR
	END_IF
	sStrHeaderLine := CONCAT(sStrHeaderLine,sLineFeed); (* concat Linefeed *)
	udiSize :=  LEN(sStrHeaderLine);
	MEMCPY( ADR(sHeader)+udiStrWriteIndex, ADR(sStrHeaderLine),udiSize);
	udiStrWriteIndex := udiStrWriteIndex + udiSize;

	(*Line: 4*)
	sStrHeaderLine 	:= '';
	sStrHeaderLine := CONCAT(sStrHeaderLine,'TurbineNumber:');
	sStrHeaderLine := CONCAT(sStrHeaderLine,sTab);
	sStrHeaderLine := CONCAT(sStrHeaderLine,UINT_TO_STRING(st_xTurbineIdent.iTurbineNumber));

	iHeaderLEN := LEN(sStrHeaderLine);
	IF iHeaderLEN < giHeaderLineLenght THEN
		FOR i := iHeaderLEN+1 TO (giHeaderLineLenght-2) DO
			sStrHeaderLine := CONCAT(sStrHeaderLine,' ');		(* concat with stuff spaces *)
		END_FOR
	END_IF
	sStrHeaderLine := CONCAT(sStrHeaderLine,sLineFeed); (* concat Linefeed *)
	udiSize :=  LEN(sStrHeaderLine);
	MEMCPY( ADR(sHeader)+udiStrWriteIndex, ADR(sStrHeaderLine),udiSize);
	udiStrWriteIndex := udiStrWriteIndex + udiSize;

	(*Line: 5*)
	sStrHeaderLine 	:= '';
	sStrHeaderLine := CONCAT(sStrHeaderLine,'TurbineType:');
	sStrHeaderLine := CONCAT(sStrHeaderLine,sTab);
	sStrHeaderLine := CONCAT(sStrHeaderLine,st_xTurbineIdent.sTurbineType);

	iHeaderLEN := LEN(sStrHeaderLine);
	IF iHeaderLEN < giHeaderLineLenght THEN
		FOR i := iHeaderLEN+1 TO (giHeaderLineLenght-2) DO
			sStrHeaderLine := CONCAT(sStrHeaderLine,' ');		(* concat with stuff spaces *)
		END_FOR
	END_IF
	sStrHeaderLine := CONCAT(sStrHeaderLine,sLineFeed); (* concat Linefeed *)
	udiSize :=  LEN(sStrHeaderLine);
	MEMCPY( ADR(sHeader)+udiStrWriteIndex, ADR(sStrHeaderLine),udiSize);
	udiStrWriteIndex := udiStrWriteIndex + udiSize;

	(*Line: 6*)
	sStrHeaderLine := '';			(* empty row *)

	iHeaderLEN := LEN(sStrHeaderLine);
	IF iHeaderLEN < giHeaderLineLenght THEN
		FOR i := iHeaderLEN+1 TO (giHeaderLineLenght-2) DO
			sStrHeaderLine := CONCAT(sStrHeaderLine,' ');		(* concat with stuff spaces *)
		END_FOR
	END_IF
	sStrHeaderLine := CONCAT(sStrHeaderLine,sLineFeed); (* concat Linefeed *)
	udiSize :=  LEN(sStrHeaderLine);
	MEMCPY( ADR(sHeader)+udiStrWriteIndex, ADR(sStrHeaderLine),udiSize);
	udiStrWriteIndex := udiStrWriteIndex + udiSize;

	(*Line: 7*)
	sStrHeaderLine 	:= '';
	(* Add description of file to the header ---------------------------*)
	sStrHeaderLine := CONCAT(sStrHeaderLine,'Comment:');
	sStrHeaderLine := CONCAT(sStrHeaderLine,sTab);
	sStrHeaderLine := CONCAT(sStrHeaderLine,s_FileDescription);

	iHeaderLEN := LEN(sStrHeaderLine);
	IF iHeaderLEN < giHeaderLineLenght THEN
		FOR i := iHeaderLEN+1 TO (giHeaderLineLenght-2) DO
			sStrHeaderLine := CONCAT(sStrHeaderLine,' ');		(* concat with stuff spaces *)
		END_FOR
	END_IF
	sStrHeaderLine := CONCAT(sStrHeaderLine,sLineFeed); (* concat Linefeed *)
	udiSize :=  LEN(sStrHeaderLine);
	MEMCPY( ADR(sHeader)+udiStrWriteIndex, ADR(sStrHeaderLine),udiSize);
	udiStrWriteIndex := udiStrWriteIndex + udiSize;

	(*Line: 8*)
	sStrHeaderLine := '';			(* first empty row *)

	iHeaderLEN := LEN(sStrHeaderLine);
	IF iHeaderLEN < giHeaderLineLenght THEN
		FOR i := iHeaderLEN+1 TO (giHeaderLineLenght-2) DO
			sStrHeaderLine := CONCAT(sStrHeaderLine,' ');		(* concat with stuff spaces *)
		END_FOR
	END_IF
	sStrHeaderLine := CONCAT(sStrHeaderLine,sLineFeed); (* concat Linefeed *)
	udiSize :=  LEN(sStrHeaderLine);
	MEMCPY( ADR(sHeader)+udiStrWriteIndex, ADR(sStrHeaderLine),udiSize);
	udiStrWriteIndex := udiStrWriteIndex + udiSize;

	(*Line: 9*)
	sStrHeaderLine := '';			(* second empty row *)

	iHeaderLEN := LEN(sStrHeaderLine);
	IF iHeaderLEN < giHeaderLineLenght THEN
		FOR i := iHeaderLEN+1 TO (giHeaderLineLenght-2) DO
			sStrHeaderLine := CONCAT(sStrHeaderLine,' ');		(* concat with stuff spaces *)
		END_FOR
	END_IF
	sStrHeaderLine := CONCAT(sStrHeaderLine,sLineFeed); (* concat Linefeed *)
	udiSize :=  LEN(sStrHeaderLine);
	MEMCPY( ADR(sHeader)+udiStrWriteIndex, ADR(sStrHeaderLine),udiSize);
	udiStrWriteIndex := udiStrWriteIndex + udiSize;

	(*Line: 10*)
	sStrHeaderLine := '';			(* third empty row *)

	iHeaderLEN := LEN(sStrHeaderLine);
	IF iHeaderLEN < giHeaderLineLenght THEN
		FOR i := iHeaderLEN+1 TO (giHeaderLineLenght-2) DO
			sStrHeaderLine := CONCAT(sStrHeaderLine,' ');		(* concat with stuff spaces *)
		END_FOR
	END_IF
	sStrHeaderLine := CONCAT(sStrHeaderLine,sLineFeed); (* concat Linefeed *)
	udiSize :=  LEN(sStrHeaderLine);
	MEMCPY( ADR(sHeader)+udiStrWriteIndex, ADR(sStrHeaderLine),udiSize);
	udiStrWriteIndex := udiStrWriteIndex + udiSize;


	(*Write to output - variable*)
	iCountsOfLine	:= 10;
	iHeaderLEN :=UDINT_TO_INT(udiStrWriteIndex);
	MEMCPY(adr_sHeader1,ADR(sHeader),udiStrWriteIndex);


(*=====================================================================*)
(*					HEADER PART 2  (column descriptions)				     *)
(*=====================================================================*)
	 (*Description with s_ColumnText, direct input string *)
	MEMSET(ADR(sColumnLine),0,SIZEOF(sColumnLine));
	udiStrWriteIndex := 0;
	IF s_ColumnText<>'' THEN
		sStrVar := CONCAT(s_ColumnText,sTab);
		iStrLEN := LEN(sStrVar);
		MEMCPY( ADR(sColumnLine)+udiStrWriteIndex, ADR(sStrVar), iStrLEN);
		udiStrWriteIndex := udiStrWriteIndex + LEN(sStrVar);
	ELSE
		sColumnLine := '';
	END_IF

	 (*Description with text out of the ARRAY, not direct - over input array*)
	FOR i:=1 TO (iCountsOfColumns) DO
		sStrVar := '';
		MEMCPY(ADR(sStrVar), ADR(ar_ColumnText[i]), SIZEOF(ar_ColumnText[i]));
		sStrVar := CONCAT(sStrVar,sTab);
		iStrLEN := LEN(sStrVar);
		MEMCPY( ADR(sColumnLine)+udiStrWriteIndex, ADR(sStrVar), iStrLEN);
		udiStrWriteIndex := udiStrWriteIndex + LEN(sStrVar);
	END_FOR

	(* fill the line to entry length  neccessarry for Statuscode !*)
	iColumnLineLEN := LEN(sColumnLine);
	IF iColumnLineLEN < iOneEntryLength THEN
		sStrVar := ' ';
		udiSize :=  LEN(sStrVar);
		FOR i := iColumnLineLEN+1 TO (iOneEntryLength-2) DO (* concat with stuff spaces *)
			MEMCPY( ADR(sColumnLine)+udiStrWriteIndex, ADR(sStrVar), udiSize);
			udiStrWriteIndex := udiStrWriteIndex + LEN(sStrVar);
		END_FOR
	END_IF

	sStrVar := sLineFeed; 	(* concat Linefeed *)
	udiSize :=  LEN(sStrVar);
	MEMCPY( ADR(sColumnLine)+udiStrWriteIndex, ADR(sStrVar),udiSize);

	(*Write to output - variable*)
	iColumnLineLEN :=LEN(sColumnLine);
	MEMCPY(adr_sColumnLine,ADR(sColumnLine),iColumnLineLEN);


(*=============== END OF FUNCTION_BLOCK / PROGRAMM =================*)

END_FUNCTION_BLOCK

// ---- Alarm System/POUs/02_Alarm_Handling/FB_WriteEventData_Day.TcPOU
FUNCTION_BLOCK FB_WriteEventData_Day
(**********************************************************************************)
(**********************************************************************************)
(*  	VERSION:			002.001
							                									
 	PROGRAMMED BY:	Puja					  					
  	Changed by:			Hardy Patommel							
*)   																		 
(*----------------------------------------------------------------------------------------------------------------------------------------------------------------*)
(*  	REVISIONS:
 	Date		|	Version/Author 	|	Remark
     ----------------------------------------------------------------------------------------------------
     	2007-04-23	|	001.001     HP		|	Error in init state by nMode -  changed to FOPEN_MODEREAD only
     	2007-10-08	|	001.002     HP		|	formatting the REAL value FOR the file output
     	2008-03-04	|	002.000     HP		|   	add header function block	
	2008-03-10	|	002.001     HP		|   	delete file enable					                									 
*)
(*----------------------------------------------------------------------------------------------------------------------------------------------------------------*)
(*  	DESCRIPTION:

*)						               				 					
(*----------------------------------------------------------------------------------------------------------------------------------------------------------------*)
VAR_INPUT
	bExecute 				: BOOL;
	sNetId					: T_AmsNetId;
	sPathName				: T_MaxString;
	dwTransferBufferStartAdr	: DWORD;
	iNewValues				: INT;
	udNumberofValues 		: UDINT;
	udNumberOfEventDatas	: UDINT;
	udArrDataSize			: ARRAY [1..NUMBER_OF_EVENT_DATAS] OF UDINT;
	eDataType				: ARRAY [1..NUMBER_OF_EVENT_DATAS] OF E_DataType;
	sHeaderOfEventData		: ARRAY [1..giGeneralLoggerChannelInUsed] OF STRING(giGeneralLenghtOfName);
END_VAR
VAR_OUTPUT
	udValuesWritten			: UDINT;
	bBusy					: BOOL;
	bDone					: BOOL;
	bError					: BOOL;
	nErrId					: UDINT;
END_VAR
VAR
	RExec_Trig				: R_TRIG;
	hFile					: UINT;
	fbFileOpen				: FB_FileOpen;
	fbFileWrite				: FB_FileWrite;
	fbFileClose				: FB_FileClose;
	tAdsTimeOut				: TIME:= T#10s;
	eFileState				: E_FileState_SC;
	nMode					: DWORD;

	sStrBuffer				: STRING(10000);
	sStrHeader				: STRING(2160);
	sVar					: STRING(255);
	sHeader					: STRING(giHeaderColumnLineLEN);
	sTab					: STRING[2] := '$T';
	sLineFeed				: STRING[4] := '$R$N';
	i						: INT;

	dwCaptureTransferBufferStartAdr : DWORD;
	sTimeStamp				: STRING[24];	(* Time the Statuscode becomes true *)
	sTrigEvent				: STRING[guiKeyAndTextLen];	(* key and Text of Statuscode, like sKeyAndText[80] in M_AddEvent*)
	sUserName				: STRING[24];	(* name of the user who had the Active Status to do the operation *)
	sBrakeProgram			: STRING[4];
	bVar 					: BOOL;
	siVar					: SINT;
	iVar						: INT;
	diVar					: DINT;
	usiVar					: USINT;
	uiVar					: UINT;
	udiVar					: UDINT;
	rVar						: REAL;
	lrVar					: LREAL;
(*	eTime					:= 12,
	eDate					:= 13,
	eTime_OF_Day			:= 14,
	eDateAndTime			:= 15,
	eString					:= 16,	*)
	byVar					: BYTE;
	wVar					: WORD;
	dwVar					: DWORD;
	strVar					: STRING;

	iCopyOffset				: INT;

	iPrepIndex				: INT;
	iStrBufferIdx				: INT; (*Index buffer*)
	iStrLineIdx				: INT; (*Index line*)
	iStuff					: INT;
	iStartStuffIndex			: INT;
	iEndStuffIndex			: INT;
	iStartIndex				: INT;
	iEndIndex				: INT;

	iBatchValue				: INT := 20;(* in batch of how many entries is the data to be written *)
	iEventsWrittenCurrent		: INT;		(* Event written in current cycle *)
	iCaptureNewValues		: INT;		(* captures new values *)
	iEventsInCycle			: INT;		(* In how many batches is data written *)
	bHeader					: BOOL;		(* If a new file write then to write the header *)
	iCounter					: INT;		(* Total number of entries written till now, so as to tally *)
	iNumberOfEventDatas		: INT;
	iEntriesWritten			: INT;
	iFileOpenedCounter		: INT;
	iFileClosedCounter		: INT;
	sTimestampShort			: STRING[12];
	sRealDataReduce		: STRING[10];
	iLength					: INT;
	iDiffenzLength				: INT;
	iForIndex					: UINT;
	fbHeaderForLogging		: FB_HeaderForLogging;
	iFirstHeaderLEN			: INT;
	iColumnLineLEN			: INT;
	iHeaderLEN				: INT;  (*length of whole header; first header + column*)
	uiCountsOfLine			: UINT;

END_VAR
VAR PERSISTENT
	nNextPointerLoc			: DINT;
END_VAR

RExec_Trig( CLK := bExecute );

CASE eFileState OF
   eInit_SC:
		IF RExec_Trig.Q THEN	(* Rising edge triggered *)
			bBusy 	:= TRUE;
			bError	:= FALSE;
			bDone 	:= FALSE;
			nErrId	:= 0;
			hFile	:= 0;
			dwCaptureTransferBufferStartAdr := dwTransferBufferStartAdr;		(* capture the transfer buffer address *)
			iCaptureNewValues	:= iNewValues;				(* make a copy of the input newvalues *)
			iNumberOfEventDatas := UDINT_TO_INT(udNumberOfEventDatas);
			nMode := FOPEN_MODEREAD OR FOPEN_MODEBINARY;
			IF  iOneEntryLength <> 0 THEN										(*Added RM2008-07-18*)
				iBatchValue := (SIZEOF(sStrBuffer)/iOneEntryLength) - 1;				(* calculate the batch size in which data is to be written *)
			END_IF
			IF iCaptureNewValues > 0 THEN
				sTimestampShort :='2';(* FUN_TimeToString(Lib_strucSystemTime); (*access time *) TO ACTION*)
				(* Open a file *)
				fbFileOpen( bExecute	:= FALSE	);
				fbFileOpen(	bExecute	:= TRUE,
							sNetId		:= sNetID,
							sPathName	:=sPathName,
							nMode		:= nMode,
							ePath		:= Path_Generic,
							tTimeout	:= tAdsTimeOut );

				eFileState := eFileOpen_SC;
				(* reset the variables *)
				iStartIndex := 1;
				iStrBufferIdx := 0;
				sStrBuffer := '';
				sVar := '';
				udValuesWritten := 0;
			END_IF
		END_IF

		g_TriggSendExeAlarmListDay := FALSE;

	eFileOpen_SC:	(* Wait for the file to be opened *)
		fbFileOpen( );
		IF NOT fbFileOpen.bBusy THEN
			fbFileOpen(	bExecute := FALSE);

			IF NOT fbFileOpen.bError THEN		(* if no error; File already exists *)

				(* calculate the minimum of Captured values, Batch value and how many can fit *)
				iEndIndex := MIN(iCaptureNewValues,iBatchValue);
				iEventsWrittenCurrent := MIN(iCaptureNewValues,iBatchValue);

				(* Close the file, nMode := FOPEN_MODEREAD *)
				fbFileClose(	bExecute:= FALSE	);
				fbFileClose(	bExecute:= TRUE,
								sNetId	:= sNetID,
								hFile	:= fbFileOpen.hFile,
								tTimeout:= tAdsTimeOut	);

				eFileState := eFileOpenExistFile_SC;

			ELSE	(*if error, File does not exist; a new file is to be written *)
				(*error by opening the file >> new file with header*)
				nMode := FOPEN_MODEAPPEND  OR FOPEN_MODEPLUS OR FOPEN_MODEBINARY;
				fbFileOpen( bExecute	:= FALSE	);
				fbFileOpen(	bExecute	:= TRUE,
							sNetId		:= sNetID,
							sPathName	:= sPathName,
							nMode		:= nMode,
							ePath		:= Path_Generic,
							tTimeout	:= tAdsTimeOut );
				iFileOpenedCounter := iFileOpenedCounter + 1;

				eFileState := eFileOpen_SC;
				iCounter := 0;
				(* if new file is being written then write down the header *)
				bHeader := TRUE;

				fbHeaderForLogging(
						st_TurbineIdent		:= st_xTurbineIdent ,		(*general machine info*)
						s_FileDescription		:= fbSCLogger.stFileSetupDayFile.sFileDescription,
						s_ColumnText 		:= gstrRingBufferFileColumnText,
						ar_ColumnText		:= sHeaderOfEventData ,	(*array of column description*)
						iCountsOfColumns		:= iNumberOfEventDatas,	(*counts of columns*)
						iOneEntryLength		:= giRingBufferFileOneEntryLength,(*length of every entry, all lines with the same length, see init-logger*)
				//ACTION		adr_sHeader1		:= ADR(sStrHeader) ,		(*part one of the header*)
				//ACTION		adr_sColumnLine		:= ADR(sHeader),			(*part two of the header*)
						iCountsOfLine			=> uiCountsOfLine,			(*lines of the part one header*)
						iHeaderLEN			=> iFirstHeaderLEN,		(*length of the part one header*)
						iColumnLineLEN		=> iColumnLineLEN);		(*length of the part two header*)

				iHeaderLEN := iFirstHeaderLEN + iColumnLineLEN;

			END_IF
		END_IF



	eFileOpenExistFile_SC:
		fbFileClose( );
		IF NOT fbFileClose.bBusy THEN
			fbFileClose(	bExecute := FALSE);
			IF NOT fbFileClose.bError THEN

				nMode := FOPEN_MODEAPPEND  OR FOPEN_MODEPLUS OR FOPEN_MODEBINARY;
				fbFileOpen( bExecute	:= FALSE	);
				fbFileOpen(	bExecute	:= TRUE,
							sNetId		:= sNetID,
							sPathName	:= sPathName,
							nMode		:= nMode,
							ePath		:= Path_Generic,
							tTimeout	:= tAdsTimeOut );
				iFileOpenedCounter := iFileOpenedCounter + 1;

				eFileState := eFileSeek_SC;
			ELSE
				bBusy := FALSE;
				bError := TRUE;
				nErrId := fbFileClose.nErrId;
				eFileState := eInit_SC;
			END_IF
		END_IF



	eFileSeek_SC:
		fbFileOpen( );
		IF NOT fbFileOpen.bBusy THEN
			fbFileOpen(	bExecute := FALSE);
			IF NOT fbFileOpen.bError THEN

				(* Prepare the data to be written *)
				M_PrepareWriteData( );

				(* Write into File *)
				fbFileWrite( 	bExecute	:= FALSE	);
				fbFileWrite(  	bExecute	:= TRUE,
								sNetId		:= sNetID,
								hFile		:= fbFileOpen.hFile,
								pWriteBuff	:= ADR(sStrBuffer),
								cbWriteLen	:= iStrBufferIdx,         (*Write not the whole Buffer, only new entries*)
								tTimeout	:= tAdsTimeOut	);
				eFileState := eFileWrite_SC;
			ELSE
				bBusy := FALSE;
				bError := TRUE;
				nErrId := fbFileOpen.nErrId;
				eFileState := eInit_SC;
			END_IF
		END_IF

	eFileWrite_SC:	(* Wait until  the file is written *)
		fbFileWrite();
		IF NOT fbFileWrite.bBusy THEN
			fbFileWrite(bExecute := FALSE);
			IF NOT fbFileWrite.bError THEN
				bHeader := FALSE;
				IF iCaptureNewValues > iEventsWrittenCurrent THEN		(* data is to be written into two or more parts *)
					IF iEventsWrittenCurrent = iBatchValue THEN
						(* sStrBuffer was insufficient to occupy all entries, Fitting entries were greater than that, continue writting at same file pointer *)
						iCaptureNewValues := iCaptureNewValues - iEventsWrittenCurrent;
						iEventsWrittenCurrent := iEndIndex := MIN( iCaptureNewValues , iBatchValue);
						iStrBufferIdx := 0;				(* reset while new batch write *)

						(* Prepare the next batch of data to be written *)
						M_PrepareWriteData( );

						(* Write into File *)
						fbFileWrite( 	bExecute	:= FALSE	);
						fbFileWrite(  	bExecute	:= TRUE,
										sNetId		:= sNetID,
										hFile		:= fbFileOpen.hFile,
										pWriteBuff	:= ADR(sStrBuffer),
										cbWriteLen	:= iStrBufferIdx,         (*Write not the whole Buffer, only new entries*)
										tTimeout	:= tAdsTimeOut	);
						eFileState := eFileWrite_SC;
					END_IF
				ELSE	(* if exact fit then reintialise pointer to start of file *)

					(* Close the File *)
					fbFileClose(	bExecute:= FALSE	);
					fbFileClose(	bExecute:= TRUE,
									sNetId	:= sNetID,
									hFile	:= fbFileOpen.hFile,
									tTimeout:= tAdsTimeOut	);
					eFileState := eFileClose_SC;
					iFileClosedCounter := iFileClosedCounter + 1;
				END_IF
			ELSE
				bBusy := FALSE;
				bError := TRUE;
				nErrId := fbFileWrite.nErrId;
				eFileState := eInit_SC;
			END_IF
		END_IF



	eFileClose_SC:	(* Wait untill File is closed *)
		fbFileClose();
		IF NOT fbFileClose.bBusy THEN
			fbFileClose( bExecute:= FALSE );
			IF NOT fbFileClose.bError THEN
				nNextPointerLoc := iEntriesWritten * iOneEntryLength;
				IF iCounter >= UDINT_TO_INT(udNumberOfValues) THEN
					iCounter := iCounter;
				END_IF
				(*eFileState := eInit_SC;*)
				eFileState := eFileCopy_SC;
				bBusy  := FALSE;
				bDone  := TRUE;
				bHeader := FALSE;
				sStrBuffer := '';
				iCaptureNewValues := 0;
				iEventsInCycle := 0;
			ELSE
				bBusy := FALSE;
				bError := TRUE;
				nErrId := fbFileClose.nErrId;
				eFileState := eInit_SC;
			END_IF
		END_IF

	eFileCopy_SC:
			g_TriggSendExeAlarmListDay := TRUE;
			eFileState := eInit_SC;

END_CASE

ACTION M_PrepareWriteData:
IF bHeader THEN
	(*Header part one*)
	MEMCPY(ADR(sStrBuffer) ,ADR(sStrHeader),iFirstHeaderLEN);
	(*Header part two, column description*)
	MEMCPY(ADR(sStrBuffer)+iFirstHeaderLEN ,ADR(sHeader),iColumnLineLEN);
	(*index for buffer entry after the header; iHeaderLEN := iFirstHeaderLEN + iColumnLineLEN;*)
	iStrBufferIdx := iHeaderLEN;
	(* Write into File *)
END_IF

(* Stuff the data to be written into a string buffer *)
FOR iPrepIndex := iStartIndex  TO iEndIndex DO	(* for loop from new index value to the number of new values *)
	iCopyOffset := (((iPrepIndex-1)+iEventsInCycle)*iOneEntrySize); (*iCopyOffset := Offset in array ringbuffer*)
	sVar := '';
	iStrLineIdx := 0; (*index for the line, function stuff line*)
	(*gets the new dataset ####################*)
	(*gets timestamp value ---------------*)
	MEMCPY(
		ADR(sTimeStamp),
		dwCaptureTransferBufferStartAdr+iCopyOffset,
		SIZEOF(sTimeStamp));
	sVar := CONCAT('',sTimeStamp);
	sVar := CONCAT(sVar,sTab);
	iCopyOffset := iCopyOffset + SIZEOF(sTimeStamp);

	(*gets trigger event string ---------------*)
	MEMCPY(
		ADR(sTrigEvent),
		dwCaptureTransferBufferStartAdr+iCopyOffset,
		SIZEOF(sTrigEvent));
	(*look and fill to 50 sign*)
	iLength := LEN(sTrigEvent);
	IF (iLength<>giCountsOfKeyLetterForStatuscodeFile) THEN
		iDiffenzLength := giCountsOfKeyLetterForStatuscodeFile - iLength ;
		FOR iForIndex := 1 TO  iDiffenzLength DO
			sTrigEvent := CONCAT(sTrigEvent,' ');
		END_FOR
	END_IF
	sTrigEvent := sTrigEvent ;
	sVar := CONCAT(sVar,sTrigEvent);
	sVar := CONCAT(sVar,sTab);
	iCopyOffset := iCopyOffset + SIZEOF(sTrigEvent); (*read data out of log-array*)

	(*gets user name string ---------------*)
	MEMCPY(
		ADR(sUserName),
		dwCaptureTransferBufferStartAdr+iCopyOffset,
		SIZEOF(sUserName));
	sVar := CONCAT(sVar,sUserName);
	sVar := CONCAT(sVar,sTab);
	iCopyOffset := iCopyOffset + SIZEOF(sUserName);

	(*gets brake program string ---------------*)
	MEMCPY(
		ADR(sBrakeProgram),
		dwCaptureTransferBufferStartAdr+iCopyOffset,
		SIZEOF(sBrakeProgram));
	sVar := CONCAT(sVar,sBrakeProgram);
	sVar := CONCAT(sVar,sTab);
	iCopyOffset := iCopyOffset + SIZEOF(sBrakeProgram);

	(*gets configuration data  value ---------------*)
	(* convert appropriate event datas into string format and concat into one string buffer *)
	FOR i := 1 TO iNumberOfEventDatas DO
		CASE eDataType[i] OF
			eBool :
				MEMCPY(ADR(bVar),dwCaptureTransferBufferStartAdr+iCopyOffset,udArrDataSize[i]);
				sVar := CONCAT(sVar,BOOL_TO_STRING(bVar));
				sVar := CONCAT(sVar,sTab);	(* append tab *)
				iCopyOffset := iCopyOffset + UDINT_TO_INT(udArrDataSize[i]);

			eSint :
				MEMCPY(ADR(siVar),dwCaptureTransferBufferStartAdr+iCopyOffset,udArrDataSize[i]);
				sVar := CONCAT(sVar,SINT_TO_STRING(siVar));
				sVar := CONCAT(sVar,sTab);	(* append tab *)
				iCopyOffset := iCopyOffset + UDINT_TO_INT(udArrDataSize[i]) ;

			eInt :
				MEMCPY(ADR(iVar),dwCaptureTransferBufferStartAdr+iCopyOffset,udArrDataSize[i]);
				sVar := CONCAT(sVar,INT_TO_STRING(iVar));
				sVar := CONCAT(sVar,sTab);	(* append tab *)
				iCopyOffset := iCopyOffset + UDINT_TO_INT(udArrDataSize[i]) ;

			eDint :
				MEMCPY(ADR(diVar),dwCaptureTransferBufferStartAdr+iCopyOffset,SIZEOF(diVar));
				sVar := CONCAT(sVar,DINT_TO_STRING(diVar));
				sVar := CONCAT(sVar,sTab);	(* append tab *)
				iCopyOffset := iCopyOffset + UDINT_TO_INT(udArrDataSize[i]) ;

			eByte :
				MEMCPY(ADR(byVar),dwCaptureTransferBufferStartAdr+iCopyOffset,udArrDataSize[i]);
				sVar := CONCAT(sVar,BYTE_TO_STRING(byVar));
				sVar := CONCAT(sVar,sTab);	(* append tab *)
				iCopyOffset := iCopyOffset + UDINT_TO_INT(udArrDataSize[i]) ;

			eWord :
				MEMCPY(ADR(wVar),dwCaptureTransferBufferStartAdr+iCopyOffset,udArrDataSize[i]);
				sVar := CONCAT(sVar,WORD_TO_STRING(wVar));
				sVar := CONCAT(sVar,sTab);	(* append tab *)
				iCopyOffset := iCopyOffset + UDINT_TO_INT(udArrDataSize[i]) ;

			eDword :
				MEMCPY(ADR(dwVar),dwCaptureTransferBufferStartAdr+iCopyOffset,udArrDataSize[i]);
				sVar := CONCAT(sVar,DWORD_TO_STRING(dwVar));
				sVar := CONCAT(sVar,sTab);	(* append tab *)
				iCopyOffset := iCopyOffset + UDINT_TO_INT(udArrDataSize[i]) ;

			eLint :
				;
	
			eUsint :
				MEMCPY(ADR(usiVar),dwCaptureTransferBufferStartAdr+iCopyOffset,udArrDataSize[i]);
				sVar := CONCAT(sVar,USINT_TO_STRING(usiVar));
				sVar := CONCAT(sVar,sTab);	(* append tab *)
				iCopyOffset := iCopyOffset + UDINT_TO_INT(udArrDataSize[i]) ;

			eUint :
				MEMCPY(ADR(uiVar),dwCaptureTransferBufferStartAdr+iCopyOffset,udArrDataSize[i]);
				sVar := CONCAT(sVar,INT_TO_STRING(iVar));
				sVar := CONCAT(sVar,sTab);	(* append tab *)
				iCopyOffset := iCopyOffset + UDINT_TO_INT(udArrDataSize[i]) ;

			eUdint :
				MEMCPY(ADR(udiVar),dwCaptureTransferBufferStartAdr+iCopyOffset,udArrDataSize[i]);
				sVar := CONCAT(sVar,UDINT_TO_STRING(udiVar));
				sVar := CONCAT(sVar,sTab);	(* append tab *)
				iCopyOffset := iCopyOffset + UDINT_TO_INT(udArrDataSize[i]) ;

			eUlint :
				;

			eReal :
				(*formatting the real value*)
				MEMCPY(ADR(rVar),dwCaptureTransferBufferStartAdr+iCopyOffset,udArrDataSize[i]);
				sRealDataReduce := '3';(*FUN_Real_to_string(rVar,2);	TO ACTION*)

				sVar := CONCAT(sVar,sRealDataReduce);
				sVar := CONCAT(sVar,sTab);	(* append tab *)
				iCopyOffset := iCopyOffset + UDINT_TO_INT(udArrDataSize[i]) ;

			eLreal :
				MEMCPY(ADR(lrVar),dwCaptureTransferBufferStartAdr+iCopyOffset,udArrDataSize[i]);
				sVar := CONCAT(sVar,LREAL_TO_STRING(lrVar));
				sVar := CONCAT(sVar,sTab);	(* append tab *)
				iCopyOffset := iCopyOffset + UDINT_TO_INT(udArrDataSize[i]) ;

			eTime :
				;

			eTime_OF_Day :
				;

			eWString :
				MEMCPY(ADR(strVar),dwCaptureTransferBufferStartAdr+iCopyOffset,udArrDataSize[i]);
				sVar := CONCAT(sVar,strVar);
				sVar := CONCAT(sVar,sTab);	(* append tab *)
				iCopyOffset := iCopyOffset + UDINT_TO_INT(udArrDataSize[i]) ;

		END_CASE
	END_FOR

	iStrLineIdx := iStrLineIdx + LEN(sVar);			(*length of string in one row*)
	iStartStuffIndex := iStrLineIdx + 1;				(*start address for stuff sign*)
	iEndStuffIndex := iOneEntryLength-2;

	(* append spaces to make every event of same length *)
	IF iStrLineIdx < iEndStuffIndex THEN
		FOR iStuff := iStartStuffIndex TO  iEndStuffIndex DO
			sVar := CONCAT(sVar,' ');
			iStrLineIdx := iStrLineIdx + 1;
		END_FOR
	END_IF
	sVar := CONCAT(sVar,sLineFeed);			(* append line feed *)
	iStrLineIdx := iStrLineIdx + LEN(sLineFeed);	(*length of string in one row*)

	(* copy the event into the string buffer *)
	IF bHeader THEN
		MEMCPY(
			ADR(sStrBuffer)+ iHeaderLEN + (iOneEntryLength * (iPrepIndex - 1)) ,
			ADR(sVar),
			iOneEntryLength);
	ELSE
		MEMCPY(
			ADR(sStrBuffer)+ (iOneEntryLength * (iPrepIndex - 1)) ,
			ADR(sVar),
			iOneEntryLength);
	END_IF
	iStrBufferIdx := iStrBufferIdx + iOneEntryLength;
	iStrLineIdx := 0;
	iCounter := iCounter + 1;


END_FOR

udValuesWritten := udValuesWritten + iEndIndex;	(* output how many values already written *)
iEventsInCycle := iEventsInCycle + iEndIndex;		(* Calculate the number of events written / in how many batches *)
END_ACTION

END_FUNCTION_BLOCK

// ---- Alarm System/POUs/02_Alarm_Handling/FB_AlarmHandler.TcPOU
FUNCTION_BLOCK FB_AlarmHandler
VAR_INPUT
	sInTimeOcc:STRING[24];
	stInTimeOcc:TIMESTRUCT;
	
END_VAR
VAR_OUTPUT
END_VAR
VAR
	i: DINT;	// index for alarm array
END_VAR
	
VAR_IN_OUT
	arrAlarms: ARRAY[*] OF ST_AlarmStructure;
END_VAR

FOR i := LOWER_BOUND(arrAlarms,1) TO UPPER_BOUND(arrAlarms,1) BY 1 DO
	
END_FOR

ACTION SetAlarms:

END_ACTION

END_FUNCTION_BLOCK

// ---- Alarm System/POUs/02_Alarm_Handling/FB_AlarmResetAccessCtrl.TcPOU
(**************************************************************************************
CopyRight Atlantis Operations UK Ltd 2015
AR500 TCS

Function Block Purpose:
Need to ensure that we have access rights controls being verified here 
even though this is also controlled by the SCADA. The Safety can also be
managed through this function block. Use the TwinCAT user level controls
to this end.

Version history: Created with TwinCat V 2.11.2248
04/08/15	V 0.01		NSM - ODT First Draft
***************************************************************************************)

FUNCTION_BLOCK FB_AlarmResetAccessCtrl
VAR_INPUT
END_VAR
VAR_OUTPUT
END_VAR
VAR
	bDummy: BOOL;
END_VAR

bDummy:=FALSE;

END_FUNCTION_BLOCK

// ---- Alarm System/POUs/02_Alarm_Handling/FB_AnalogueAlarm.TcPOU
FUNCTION_BLOCK FB_AnalogueAlarm
VAR_INPUT
	fIn: LREAL;
	bLessThan: BOOL;
END_VAR
VAR_OUTPUT
END_VAR
VAR
	bAlarmActive: BOOL;
	iLT_Counter: UINT;
	iGT_Counter: UINT;
END_VAR
VAR_IN_OUT
	stAlarmStruct:ST_AlarmStructure;
END_VAR

IF bLessThan THEN

	IF fIn < stAlarmStruct.Param1.Set AND NOT stAlarmStruct.b THEN
		bAlarmActive := TRUE;

	ELSIF 	(fIn >= stAlarmStruct.Param1.Set AND NOT stAlarmStruct.b) OR
			(fIn >= stAlarmStruct.Param2.Set AND stAlarmStruct.b) THEN
		bAlarmActive := FALSE;

	END_IF

	iLT_Counter := iLT_Counter + 1;

ELSIF NOT bLessThan THEN

	IF fIn > stAlarmStruct.Param1.Set AND NOT stAlarmStruct.b THEN
		bAlarmActive := TRUE;

	ELSIF 	(fIn <= stAlarmStruct.Param1.Set AND NOT stAlarmStruct.b) OR
			(fIn <= stAlarmStruct.Param2.Set AND stAlarmStruct.b) THEN
		bAlarmActive := FALSE;

	END_IF

	iGT_Counter := iGT_Counter + 1;

END_IF

stAlarmStruct.a := bAlarmActive;

END_FUNCTION_BLOCK

// ---- Alarm System/POUs/02_Alarm_Handling/FB_MakeLoggString.TcPOU
FUNCTION_BLOCK FB_MakeLoggString
(*=================================================================================================*)
(*
	VERSION:				01.02
	PROGRAMMED BY:		RM					DATE:  2007-09-26 
	REVISED BY:				RM					DATE:  2007-12-10	

	Date		|	Version/Author 		|	Remark
	----------------------------------------------------------------------------------------------------
	2009-08-09	|	001.02     HP		|	change length of sTimeStamp[24], sText[120]	

	DESCRIPTION:		
*)
(*=================================================================================================*)

VAR_INPUT
	EventKey:		STRING[11];
	TextInfo: 			STRING[50];
END_VAR
VAR_OUTPUT
	LogText:			STRING [120];
END_VAR
VAR
	sKey:		 	STRING[12];
	iPower: 			INT;
	iFlowSpeed: 		INT;
	iGenSpeed: 		INT;
	iPitchAngle: 		INT;
	sText: 			STRING [120];
	sPower: 			STRING [4];
	sFlowSpeed: 	STRING [4];
	sGenSpeed: 		STRING [5];
	sPitchAngle: 		STRING [4];
	sTimeStamp:		STRING[24];
END_VAR

(*=============== START OF FUNCTION_BLOCK / PROGRAMM ===============*)

(*===========================================================================*)
(*  			Preparing the additional information which will be added 					*)
(*===========================================================================*)
(*	iPower:=					REAL_TO_INT (Lib_rGeneratorPower);
	iFlowSpeed:=			REAL_TO_INT (Lib_rFlowSpeed * 10);
	iGenSpeed:=				REAL_TO_INT (Lib_rGeneratorSpeed * 100);
	iPitchAngle:=				REAL_TO_INT (Lib_rPitchAngle * 10);
	sTimeStamp:=			Lib_sLocalTime;

	sPower:=			INT_TO_STRING (iPower);				(*to get for the entry a fixed number of characters *)
		IF iPower < 10 THEN
			sPower:= CONCAT('___', sPower);
		ELSIF iPower < 100 THEN
			sPower:= CONCAT('__', sPower);
		ELSIF iPower < 1000 THEN
			sPower:= CONCAT('_', sPower);
		END_IF

	sFlowSpeed:=	INT_TO_STRING (iFlowSpeed);			(*to get for the entry a fixed number of characters *)
		IF iFlowSpeed < 10 THEN
			sFlowSpeed:= CONCAT('___', sFlowSpeed);
		ELSIF iFlowSpeed < 100 THEN
			sFlowSpeed:= CONCAT('__', sFlowSpeed);
		ELSIF iFlowSpeed < 1000 THEN
			sFlowSpeed:= CONCAT('_', sFlowSpeed);
		END_IF

	sGenSpeed:=		INT_TO_STRING (iGenSpeed);			(*to get for the entry a fixed number of characters *)
		IF iGenSpeed < 10 THEN
			sGenSpeed:= CONCAT('___', sGenSpeed);
		ELSIF iGenSpeed < 100 THEN
			sGenSpeed:= CONCAT('__', sGenSpeed);
		ELSIF iGenSpeed < 1000 THEN
			sGenSpeed:= CONCAT('_', sGenSpeed);
		END_IF

	sPitchAngle:=		INT_TO_STRING (iPitchAngle);			(*to get for the entry a fixed number of characters *)
		IF iPitchAngle < 10 THEN
			sPitchAngle:= CONCAT('___', sPitchAngle);
		ELSIF iPitchAngle < 100 THEN
			sPitchAngle:= CONCAT('__', sPitchAngle);
		ELSIF iPitchAngle < 1000 THEN
			sPitchAngle:= CONCAT('_', sPitchAngle);
		END_IF
*)
	sTimeStamp:=	Lib_sLocalTime;
	sPower:= 		REAL_TO_STRING(Lib_rGeneratorPower);
	sFlowSpeed:= 	REAL_TO_STRING(Lib_rFlowSpeed);
	sGenSpeed:= 	REAL_TO_STRING(Lib_rGeneratorSpeed);
(*	sPitchAngle:= 	REAL_TO_STRING(Lib_rPitchAngle);	*)

(*===========================================================================*)
(* 					Putting together the String for logging							*)
(*===========================================================================*)
	sKey := CONCAT ( MID(EventKey, 9, 3),'   '); 	(*9+1*)

	sText := CONCAT(sTimeStamp,'  ');  			(*24*)
	sText := CONCAT(sText, sPower);			(*5*)
	sText := CONCAT(sText,'  ');
	sText := CONCAT(sText, sFlowSpeed);		(*5*)
	sText := CONCAT(sText,'  ');
	sText := CONCAT(sText, sGenSpeed);		(*5*)
	sText := CONCAT(sText,'  ');
	sText := CONCAT(sText, sPitchAngle);  		(*5*)

	sText := CONCAT(sText,'  ');
	sText := CONCAT(sText, sKey); 				(*12*)
	sText := CONCAT(sText,'  ');
	sText := CONCAT(sText, TextInfo); (*summary 56 + 12 + 50 >> 118*)

(*===========================================================================*)
(*						Copy to VAR_OUTPUT								*)
(*===========================================================================*)
	LogText:= sText;

(*========== END OF FUNCTION_BLOCK / PROGRAMM ======================*)

END_FUNCTION_BLOCK

// ---- Alarm System/POUs/02_Alarm_Handling/PRG_MAIN_StatuscodeLogger.TcPOU
PROGRAM PRG_MAIN_StatuscodeLogger
(**********************************************************************************)
(**********************************************************************************)
(*  	VERSION:				001.001

  	PROGRAMMED BY:		Robert Müller
  	Changed BY:				
	DATE:					2009-10-30
*)							               				 			
(*-------------------------------------------------------------------------------------------------------*)
 (*  	REVISIONS:
   	Date		|	Version/Author 		|	Remark
	----------------------------------------------------------------------------------------------------
	2009-10-30	|	001.001     RM			|	Prepared for Library
       									 
*)
(*--------------------------------------------------------------------------------------------------------*)
(*  	DESCRIPTION:

*)
(**********************************************************************************)
(**********************************************************************************)
VAR_INPUT
	TriggStatuscode:	BOOL;
	SendAlarm:		BOOL;
	EventKey:		STRING[11];
	TextInfo:			STRING[50];
	UserName:		STRING[24];
	BrakeProgram: STRING[4];
	PathNamePC:		T_MaxString;
	PathNameEmbPC:	T_MaxString;
	DailyFile:		BOOL;
	FreezeList :		BOOL;
	SCandOC:		BOOL;

	CheckLog:		BOOL;
	ResetErrCnt:		BOOL;
END_VAR
VAR_OUTPUT
	Error:	BOOL;
	iErrCounter:	UDINT;
END_VAR
VAR
	rTriggSC: 			R_TRIG;
	fbHeaderForLogging: 	FB_HeaderForLogging;

	bInitDone: 			BOOL ;
	iFirstHeaderLEN: 		INT;
	iColumnLineLEN: 		INT;

	fbF_TRIG: F_TRIG;

	bInitComplete: BOOL;			(*Inhibits status code logger until the init is complete*)


(*	fbToggle: FB_Toggle;	*)
END_VAR

(*========== START OF FUNCTION_BLOCK / PROGRAMM ============*)

(* INHIBIT SC  LOGGER UNTIL INIT COMPLETE - 09/02/17  AG. *)
fbF_TRIG(CLK:=g_bOperMaStInitSt);

IF fbF_TRIG.Q THEN
	bInitComplete:=TRUE;
END_IF
(*fbToggle(bEnable:=TRUE , tOffDelay:=T#80ms, tOnDelay:=T#10ms , bToggle=>);	*)
(*=======================================================================*)
(*			INIT  LOGGING			    									*)
(*=======================================================================*)
	IF NOT bInitDone THEN

		M_InitLoggerStatuscodes();			(*Initializing the header and the path name*)
		bInitDone:=	TRUE;

(*===========================================================================*)
(* 				General information for rising and falling edge of Statuscode 			*)
(*===========================================================================*)
	ELSE
		fbSCLogger(
			bWriteDayFile:=  DailyFile);

		rTriggSC (CLK:=	TriggStatuscode );


	(*===========================================================================*)
	(*   			RINGBUFFER for Statuscodes / BUFFER  for Sending Alarms			*)
	(*===========================================================================*)

		IF rTriggSC.Q THEN

			(*Logger for logging on PLC hard disc:  _____________________________*)
			fbSCLogger.M_AddEvent(
					bTrigEvent 			:= TRUE ,
					sTimeStamp			:= gsLocalSystemTime,
					sTrigEventKey		:= EventKey,							(* Key of the Statuscode *)
					sTrigEventText		:= TextInfo,							(* Name / Description of the Statuscode *)
					sUserName			:= UserName,							(* User name who owns access rights*)
					sBrakeProgram		:= BrakeProgram,					(* Brake program *)

					bWriteDayFile		:= DailyFile,
					CheckLog			:= CheckLog,
					ResetErrCnt			:= ResetErrCnt,

					bError=>				Error,
					nErrID=>				iErrCounter);




			(*Log List for sending alarms:  _____________________________________ POISTETTU KÄYTÖSTÄ TURHANA??? MLe*)
			(*IF SendAlarm THEN

				PRG_SendBuffAlarms( 	EventKey:=		EventKey,
									TextInfo:= 		TextInfo);
			END_IF POISTA*)


		END_IF

	END_IF

(*=========== END OF FUNCTION_BLOCK / PROGRAMM =============*)

ACTION M_InitLoggerStatuscodes:
(*    START OF METHOD   ( M_InitLoggerStatuscodes) 			*)
(*======================================================	*)

(********************************************************************************************)

(*  	VERSION:			002.001
							                									 
  	PROGRAMMED BY:	Hardy Patommel		  					
  	DATE:				2008-03-04
*)							               				 					
(*---------------------------------------------------------------------------------------------------*)
	(* Version history:
	Date		|	Version/Author 		|	Remark
	----------------------------------------------------------------------------------------------------
	2008-03-04	|	001.000     HP			|	
 	2009-10-30	|	002.001 RM			|	Prepared for Library
						                									 
*)
(*-----------------------------------------------------------------------------------------------------*)
(*  	DESCRIPTION:		Initialisations of all basic information for the
						Statuscode logger (for writing the log to a file on hard disc)

	NOTE:				the path / directory  information depends on
						which hardware and which operating system the
						project is running. That's important, when you will run the 
						software not only on the real target system but for testing  
						also on your office PC or any other PC
*)
(********************************************************************************************)

	(* Set the Path name:   ----------------------------------------------------- *)
	IF NOT gbOperatingSystemCEDetected THEN
		gsSC_PathName			:= DirectoriesFiles.sSC_PathNamePC;
(*		gsSCunlimited_PathName 	:= gsSCunlimited_PathNamePC;	*)

	ELSE
		gsSC_PathName			:= DirectoriesFiles.sSC_PathNameEmbeddedPC;
(*		gsSCunlimited_PathName	:= gsSCunlimited_PathNameEmbeddedPC;	*)
	END_IF

	(* Ringbuffer File setup  ---------------------------------------------------- *)
	fbSCLogger.stFileSetup.sNetId 				:= '';					(* Set the NetId *)
	fbSCLogger.stFileSetup.sPathName 		:= gsSC_PathName;		(* Set the Path name *)
	fbSCLogger.stFileSetup.sFileDescription 	:= 'Statuscode ring buffer file';

	(* Buffer File setup for Day-File  ---------------------------------- *)
	fbSCLogger.stFileSetupDayFile.sNetId 		:= '';					(* Set the NetId *)

	(* Path name with File name include the date*)
	fbSCLogger.stFileSetupDayFile.sPathName 		:=  '3';(*FUN_DateFileNameWithSpace(gsSC_PathName, Lib_strucSystemTime,'') ;	(* New Path name with date *)	ACTION*)
	fbSCLogger.stFileSetupDayFile.sPathName 		:=  CONCAT(fbSCLogger.stFileSetupDayFile.sPathName,'  ') ;	(* add space *)
	fbSCLogger.stFileSetupDayFile.sName			:= 'BufferStatuscodes.txt';
	fbSCLogger.stFileSetupDayFile.sTotalName		:=  CONCAT(fbSCLogger.stFileSetupDayFile.sPathName,fbSCLogger.stFileSetupDayFile.sName);
	fbSCLogger.stFileSetupDayFile.sFileDescription  	:= 'Statuscode file for one day';

//ACTION	fbSCLogger.dwLoggedEventAdr	:= ADR(arLoggedSC);		(* Adress of buffer where the logged events are to be stored *)
	fbSCLogger.udLoggedEventSize := SIZEOF(arLoggedSC);	(* sizeof buffer where the logged events are to be stored *)

	fbSCLogger.udNumberOfEventDatas	:= 4;

	(* Init used data, size and address*)
	fbSCLogger.eDataType[1]			:= eReal;
//ACTION	fbSCLogger.dwArrDataAdr[1] 		:= ADR(Lib_rGeneratorPower);				(* Power *)
	fbSCLogger.udArrDataSize[1] 		:= SIZEOF(Lib_rGeneratorPower);
	fbSCLogger.sHeaderOfEventData[1]	:= 'GeneratorPower';

	fbSCLogger.eDataType[2]			:= eReal;
//ACTION	fbSCLogger.dwArrDataAdr[2] 		:= ADR(Lib_rFlowSpeed);					(* FlowSpeed *)
	fbSCLogger.udArrDataSize[2] 		:= SIZEOF(Lib_rFlowSpeed);
	fbSCLogger.sHeaderOfEventData[2]	:= 'FlowSpeed';
	
	fbSCLogger.eDataType[3] 			:= eReal;
//ACTION	fbSCLogger.dwArrDataAdr[3] 		:= ADR(Lib_rGeneratorSpeed);				(* GenSpeed *)
	fbSCLogger.udArrDataSize[3] 		:= SIZEOF(Lib_rGeneratorSpeed);
	fbSCLogger.sHeaderOfEventData[3] 	:= 'GeneratorSpeed';

(*	fbSCLogger.eDataType[4] 			:= eReal;
	fbSCLogger.dwArrDataAdr[4] 		:= ADR(Lib_rPitchAngle);					(* Pitch Angle *)
	fbSCLogger.udArrDataSize[4] 		:= SIZEOF(Lib_rPitchAngle);
	fbSCLogger.sHeaderOfEventData[4] 	:= 'PitchAngle';	*)


	(*=====================================================================*)
	(*					make header only for the length account				     *)
	(*=====================================================================*)
	giRingBufferFileOneEntryLength := 100;(*Length of one entry in the ring buffer Statuscode file*)
	gstrRingBufferFileColumnText :=  '$TTrigKey$TUserName$TBrakeProgram';

	fbHeaderForLogging(
			st_TurbineIdent		:= st_xTurbineIdent ,		(*general machine info*)
			s_FileDescription		:= fbSCLogger.stFileSetup.sFileDescription,
			s_ColumnText 		:= gstrRingBufferFileColumnText,
			ar_ColumnText		:= fbSCLogger.sHeaderOfEventData,	(*array of column description*)
			iCountsOfColumns		:= UDINT_TO_INT(fbSCLogger.udNumberOfEventDatas),	(*counts of columns*)
			iOneEntryLength		:= giRingBufferFileOneEntryLength,(*length of every entry, all lines with the same length, see init-logger*)
			adr_sHeader1		:=  ,						(*part one of the header*)
			adr_sColumnLine		:=  ,						(*part two of the header*)
			iCountsOfLine			=> ,						(*lines of the part one header*)
			iHeaderLEN			=> iFirstHeaderLEN,		(*length of the part one header*)
			iColumnLineLEN		=> iColumnLineLEN);		(*length of the part two header*)

	giRingBufferFileHeaderLEN := iFirstHeaderLEN + iColumnLineLEN;

(*===============  END OF METHOD  ==========================================*)
END_ACTION

END_PROGRAM

// ---- Alarm System/POUs/02_Alarm_Handling/P_ScadaAlarmsMapping.TcPOU
PROGRAM P_ScadaAlarmsMapping
VAR
		i: UINT;
END_VAR


FOR i := 1 TO iMaxAlarms DO

	arrScadaAlarms[i].b := BOOL_TO_INT ( arrAlarms[i].b );

END_FOR

END_PROGRAM

// ---- Alarm System/POUs/02_Alarm_Handling/StatusCodes/PRG_TranslatorVarNames.TcPOU
PROGRAM PRG_TranslatorVarNames
VAR_INPUT
	rGeneratorPower:		REAL;
	rGeneratorSpeed:		REAL;
	rFlowSpeed:			REAL;
(*	rPitchAngle:			REAL;	*)

	sOffsetUTC: 			STRING[20];
	LibIniActive:			BOOL;

END_VAR
VAR_OUTPUT
	sLocalTime:			STRING[24];
	sTimeZoneInfo:		STRING[20];
	strucSystemTime:		TIMESTRUCT;

	bDetectNewYear	:	BOOL;
	bDetectNewMonth:	BOOL;
	bDetectNewDay	:	BOOL;
	bDetectNewHour	:	BOOL;
	bDetectNew10min:	BOOL;
	bDetectNew5min	:	BOOL;
	bDetectNewMinute:	BOOL;
	bDetectNew30sec:	BOOL;
	bDetectNewSecond:	BOOL;
	bDetectNew100ms:	BOOL;
END_VAR

(*========== START OF FUNCTION_BLOCK / PROGRAMM ============*)

(*===========================================================================*)
(* 		Just translating the names of in the library multiple used project variables 		*)
(*===========================================================================*)

	(*Copy VAR_INPUT to Library Variables:   -------------------------------------------*)
	Lib_rGeneratorPower:=		rGeneratorPower;
	Lib_rGeneratorSpeed:=	rGeneratorSpeed;
	Lib_rFlowSpeed:=			rFlowSpeed;
(*	Lib_rPitchAngle:=			rPitchAngle;	*)

	Lib_sOffsetUTC:=			sOffsetUTC;
	LibIniActive:=				gbInitializationActive;

	(*Copy Library Variables to VAR_OUTPUT :   -------------------------------------------*)
	sLocalTime:=			Lib_sLocalTime;
	sTimeZoneInfo:=		Lib_sOffsetUTC;
	strucSystemTime:=	Lib_strucSystemTime;

	bDetectNewYear:=	LibDetectNewYear;
	bDetectNewMonth:=	LibDetectNewMonth;
	bDetectNewDay:=		LibDetectNewDay;
	bDetectNewHour:=	LibDetectNewHour;
	bDetectNew10min:=	LibDetectNew10min;
	bDetectNew5min:=	LibDetectNew5min;
	bDetectNewMinute:=	LibDetectNewMinute;
	bDetectNew30sec:=	LibDetectNew30sec;
	bDetectNewSecond:=	LibDetectNewSecond;
	bDetectNew100ms:=	LibDetectNew100ms;


(*=========== END OF FUNCTION_BLOCK / PROGRAMM =============*)

END_PROGRAM

// ---- Alarm System/TC3 EventLogger/AlarmWithCustomSourceInfo.TcPOU
PROGRAM AlarmWithCustomSourceInfo
VAR
    bIsInitalized : BOOL;
    fbAlarm : FB_TcAlarm;
    bRaiseAlarm : BOOL;
    bClearAlarm : BOOL;
	bConfirmAlarm:BOOL; 
    fbSourceInfo : FB_TcSourceInfo;
END_VAR

IF NOT bIsInitalized THEN
    bIsInitalized := TRUE;
    fbSourceInfo.Clear();
    fbSourceInfo.sName := 'Water pump 3';
    fbAlarm.CreateEx(TC_Events.AlarmSystem.B99, FALSE, fbSourceInfo);
	
END_IF

IF bRaiseAlarm THEN
    bRaiseAlarm := FALSE;
    fbAlarm.ipArguments.Clear().AddString('Bob');
    fbAlarm.Raise(0);
END_IF

IF bConfirmAlarm THEN
    bConfirmAlarm := FALSE;
    fbAlarm.Confirm(0);
END_IF

IF bClearAlarm THEN
    bClearAlarm := FALSE;
    fbAlarm.Clear(0, TRUE);
END_IF

END_PROGRAM

// ---- Alarm System/TC3 EventLogger/OtherAlarmsWithCustomSource.TcPOU
PROGRAM OtherAlarmsWithCustomSource
VAR
    bIsInitalized : BOOL;
    fbAlarm : FB_TcAlarm;
    bRaiseAlarm : BOOL;
    bClearAlarm : BOOL;
	bConfirmAlarm:BOOL; 
    fbSourceInfo : FB_TcSourceInfo;
END_VAR

IF NOT bIsInitalized THEN
    bIsInitalized := TRUE;
    fbSourceInfo.Clear();
    fbSourceInfo.sName := 'Water pump 3';
    fbAlarm.CreateEx(TC_Events.NewEventClass.Event, FALSE, fbSourceInfo);
END_IF

IF bRaiseAlarm THEN
    bRaiseAlarm := FALSE;
    fbAlarm.ipArguments.Clear().AddString('Bob');
    fbAlarm.Raise(0);
END_IF

IF bConfirmAlarm THEN
    bConfirmAlarm := FALSE;
    fbAlarm.Confirm(0);
END_IF

IF bClearAlarm THEN
    bClearAlarm := FALSE;
    fbAlarm.Clear(0, TRUE);
END_IF

END_PROGRAM

// ---- Base/Devices/POU/fbMotorisedCB.TcPOU
FUNCTION_BLOCK fbMotorisedCB
VAR_INPUT
END_VAR
VAR_OUTPUT
END_VAR
VAR
END_VAR
VAR_IN_OUT
	
END_VAR

END_FUNCTION_BLOCK

// ---- Base/General Control/POU/FB_TagAlarmProps.TcPOU
FUNCTION_BLOCK FB_TagAlarmProps
VAR_INPUT
	sInTimeOcc:STRING[24];
	stInTimeOcc:TIMESTRUCT;
	bInAlarm:BOOL;
	rInturbineStatus:ST_ProcessVariables;
END_VAR
VAR_OUTPUT
	sOutTimeOcc:STRING[24];
	stOutTimeOcc:TIMESTRUCT;
	rOutturbineStatus:ST_ProcessVariables;
END_VAR
VAR
END_VAR

IF bInAlarm THEN
	sOutTimeOcc:=sInTimeOcc;
	stOutTimeOcc:=stInTimeOcc;
	rOutturbineStatus.fFlowSpeed:=rInturbineStatus.fFlowSpeed;
	rOutturbineStatus.fGeneratorSpeed:=rInturbineStatus.fGeneratorSpeed;
	rOutturbineStatus.fPitchAngle:=rInturbineStatus.fPitchAngle;
	rOutturbineStatus.fPower:=rInturbineStatus.fPower;
END_IF

END_FUNCTION_BLOCK

// ---- Base/Process Control/POU/fb2dLookup.TcPOU
FUNCTION_BLOCK fb2dLookup
VAR_INPUT
    x : REAL; (* Input value for the x-axis *)
    y : REAL; (* Input value for the y-axis *)
    table : ARRAY [1..20, 1..20] OF REAL; (* 2-D lookup table *)
END_VAR
VAR_OUTPUT
    result : REAL; (* Output value from the lookup table *)
END_VAR
VAR
    i : INT; (* Index variable for the rows *)
    j : INT; (* Index variable for the columns *)
    x_low : REAL; (* Lower boundary of x-axis interval *)
    x_high : REAL; (* Upper boundary of x-axis interval *)
    y_low : REAL; (* Lower boundary of y-axis interval *)
    y_high : REAL; (* Upper boundary of y-axis interval *)
    x_index : INT; (* Index of the x-axis interval *)
    y_index : INT; (* Index of the y-axis interval *)
    x_factor : REAL; (* Interpolation factor for x-axis *)
    y_factor : REAL; (* Interpolation factor for y-axis *)
    fx1 : REAL; (* Value at lower boundary of x-axis interval *)
    fx2 : REAL; (* Value at upper boundary of x-axis interval *)
    fy1 : REAL; (* Value at lower boundary of y-axis interval *)
    fy2 : REAL; (* Value at upper boundary of y-axis interval *)
END_VAR

(* Find the x-axis interval *)
    x_index := 1;
    FOR i := 1 TO 20 DO
        IF x >= table[i, 1] THEN
            x_index := i;
        ELSE
            EXIT;
        END_IF
    END_FOR
    
    (* Find the y-axis interval *)
    y_index := 1;
    FOR j := 1 TO 20 DO
        IF y >= table[1, j] THEN
            y_index := j;
        ELSE
            EXIT;
        END_IF
    END_FOR
    
    (* Calculate the interpolation factors *)
    x_low := table[x_index, 1];
    x_high := table[x_index+1, 1];
    y_low := table[1, y_index];
    y_high := table[1, y_index+1];
    x_factor := (x - x_low) / (x_high - x_low);
    y_factor := (y - y_low) / (y_high - y_low);
    
    (* Perform the 2-D interpolation *)
    fx1 := table[x_index, y_index] + (table[x_index+1, y_index] - table[x_index, y_index]) * x_factor;
    fx2 := table[x_index, y_index+1] + (table[x_index+1, y_index+1] - table[x_index, y_index+1]) * x_factor;
    fy1 := fx1 + (fx2 - fx1) * y_factor;
    fx1 := table[x_index+1, y_index] + (table[x_index+1, y_index+1] - table[x_index+1, y_index]) * x_factor;
    fx2 := table[x_index+1, y_index] + (table[x_index+1, y_index+1] - table[x_index+1, y_index]) * x_factor;
    fy2 := fx1 + (fx2 - fx1) * y_factor;
    result := fy1 + (fy2 - fy1) * x_factor;

END_FUNCTION_BLOCK

// ---- Base/Process Control/POU/fbRateCalc.TcPOU
FUNCTION_BLOCK fbRateCalc
FUNCTION_BLOCK Derivative
VAR_INPUT
    ProcessValue : REAL; (* The process value to calculate the derivative for *)
    SamplingPeriod : TIME := T#1S; (* The time between samples, default is 1 second *)
    AveragingPeriod : TIME := T#10S; (* The time period over which to average the samples, default is 10 seconds *)
END_VAR
VAR_OUTPUT
    Derivative : REAL; (* The calculated derivative value *)
END_VAR
VAR
    SampleTimes : ARRAY [1..10] OF TIME := [T#0S, T#0S, T#0S, T#0S, T#0S, T#0S, T#0S, T#0S, T#0S, T#0S]; (* The times at which each sample was taken *)
    Samples : ARRAY [1..10] OF REAL := [0.0, 0.0, 0.0, 0.0, 0.0, 0.0, 0.0, 0.0, 0.0, 0.0]; (* The sample values *)
    SampleIndex : INT := 0; (* The index of the current sample in the sample arrays *)
    SampleCount : INT := 0; (* The number of samples taken so far *)
    SampleSum : REAL := 0.0; (* The sum of all samples *)
    LastSampleTime : TIME := T#0S; (* The time at which the last sample was taken *)
END_VAR


(* Calculate the derivative *)
IF SampleCount > 1 THEN
    Derivative := (Samples[SampleIndex] - Samples[(SampleIndex - 1) MOD 10]) / TIME_TO_REAL(SampleTimes[SampleIndex] - SampleTimes[(SampleIndex - 1) MOD 10]);
ELSE
    Derivative := 0.0;
END_IF

(* Update the sample arrays *)
SampleIndex := (SampleIndex MOD 10) + 1;
SampleTimes[SampleIndex] := LastSampleTime;
Samples[SampleIndex] := ProcessValue;
SampleCount := SampleCount + 1;

IF SampleCount > 10 THEN
    SampleSum := SampleSum - Samples[(SampleIndex + 1) MOD 10] + ProcessValue;
ELSE
    SampleSum := SampleSum + ProcessValue;
END_IF

(* Update the averaging period *)
IF TIME_TO_REAL(LastSampleTime - SampleTimes[(SampleIndex - 1) MOD 10]) >= TIME_TO_REAL(AveragingPeriod) THEN
    Derivative := SampleSum / REAL_TO_DWORD(TIME_TO_REAL(LastSampleTime - SampleTimes[(SampleIndex - 1) MOD 10]));
    SampleSum := ProcessValue;
    SampleCount := 1;
END_IF

(* Update the last sample time *)
LastSampleTime := LastSampleTime + SamplingPeriod;

END_FUNCTION_BLOCK

// ---- Base/Resource/fbHMIBit.TcPOU
FUNCTION_BLOCK fbHMIBit
VAR_INPUT
	bInToggle:BOOL:
	bInLatch:BOOL;
END_VAR
VAR_OUTPUT
END_VAR
VAR
	RTrigHMI:R_TRIG;
END_VAR
VAR_IN_OUT
	bHMI:BOOL;
	bPLC:BOOL;
END_VAR

RTrigHMI(CLK:=bHMI , Q=> );

IF bIntoggle:BOOL:	
	IF RTrigHMI.Q AND NOT bPLC THEN
		bPLC:=1;
	END_IF
	
	IF   RTrigHMI.Q AND bPLC THEN
		bPLC:=0;
	END_IF
ELSE
	bPLC:=bHMI;
END_IF

END_FUNCTION_BLOCK

// ---- GlobalTextList.TcGTLO
TEXTLIST GlobalTextList
  202 = 'ON'
END_TEXTLIST

// ---- VISUs/Visualization.TcVIS
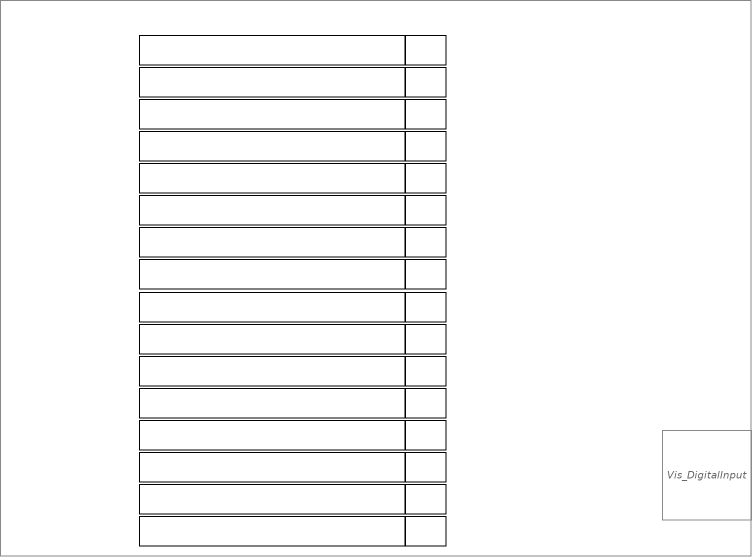
VISUALIZATION Visualization  // 752x557
    Frame (121,27 350x530)
        shows Vis_Interlock_base(stHMIInterlock := HMI.stTest01_Intlk)
    Frame (662,430 90x90)
        shows Vis_DigitalInput(stHMI_DigitalInput := HMI.stTest04_DigitalInput)
END_VISUALIZATION

// ---- VISUs/Vis_AnalogueOutput_Symbol.TcVIS
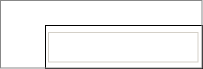
VISUALIZATION Vis_AnalogueOutput_Symbol  // 203x69
VAR_IN_OUT
	stHMI_AnalogueOutput:stHMI_AnalogueOutput;;
END_VAR
    Rectangle (45,25 158x44), colour toggle: NOT(stHMI_AnalogueOutput.bInterlock)
    Textfield (48,32 150x30), text variable: stHMI_AnalogueOutput.rValue
END_VISUALIZATION

// ---- VISUs/Vis_DigitalInput_1.TcVIS
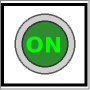
VISUALIZATION Vis_DigitalInput_1  // 90x90
VAR_IN_OUT
	stHMI_DigitalInput:stHMI_DigitalInput;
END_VAR
    Rectangle (1,3 86x83)
        p3092690914: stHMI_DigitalInput.iMode=2
    Lamp1 (10,9 70x70), style: Lamp-Lamp1-Gray
    Lamp1 (10,9 70x70), invisible if: stHMI_DigitalInput.bOn=0, style: Lamp-Lamp1-Green
    Label (16,31 56x28), "ON", invisible if: stHMI_DigitalInput.bOn=0
END_VISUALIZATION

// ---- VISUs/Vis_DigitalInput_2.TcVIS
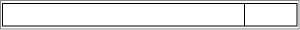
VISUALIZATION Vis_DigitalInput_2  // 300x30
VAR_IN_OUT
	stHMI_DigitalInput:stHMI_DigitalInput;
END_VAR
    Rectangle (2,3 243x23)
    Rectangle (244,3 53x23)
END_VISUALIZATION

// ---- VISUs/Vis_Interlock_base.TcVIS
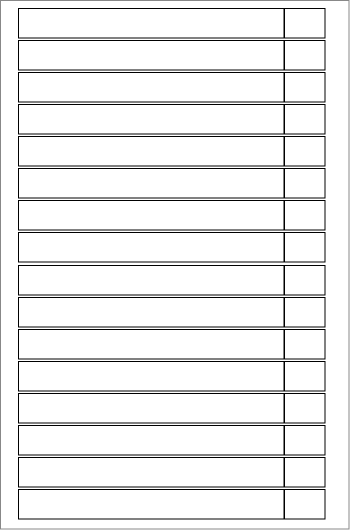
VISUALIZATION Vis_Interlock_base  // 350x530
VAR_IN_OUT
	stHMIInterlock:stHMI_Interlock;
END_VAR
    Rectangle (18,8 266x30), text variable: stHMIInterlock.asInterlockNames[1]
    Rectangle (284,8 41x30), colour toggle: stHMIInterlock.abInterlocks[1]
    Rectangle (18,40 266x30)
    Rectangle (284,40 41x30)
    Rectangle (18,72 266x30)
    Rectangle (284,72 41x30)
    Rectangle (18,104 266x30)
    Rectangle (284,104 41x30)
    Rectangle (18,136 266x30)
    Rectangle (284,136 41x30)
    Rectangle (18,168 266x30)
    Rectangle (284,168 41x30)
    Rectangle (18,200 266x30)
    Rectangle (284,200 41x30)
    Rectangle (18,232 266x30)
    Rectangle (284,232 41x30)
    Rectangle (18,265 266x30)
    Rectangle (284,265 41x30)
    Rectangle (18,297 266x30)
    Rectangle (284,297 41x30)
    Rectangle (18,329 266x30)
    Rectangle (284,329 41x30)
    Rectangle (18,361 266x30)
    Rectangle (284,361 41x30)
    Rectangle (18,393 266x30)
    Rectangle (284,393 41x30)
    Rectangle (18,425 266x30)
    Rectangle (284,425 41x30)
    Rectangle (18,457 266x30)
    Rectangle (284,457 41x30)
    Rectangle (18,489 266x30)
    Rectangle (284,489 41x30)
END_VISUALIZATION
